(* CODESYS project SPT_Base_Types.library
   Version: 4.0.4
   Title: SPT Base Types
   DefaultNamespace: SPT_BaseTypes
   Placeholder: SPT Base Types
   Company: Beckhoff Automation LLC

Project tree, tasks and I/O mapping:
  libraries: SPT Event Logger, * (Beckhoff Automation LLC); Tc2_EtherCAT, * (Beckhoff Automation GmbH); Tc2_Standard, * (Beckhoff Automation GmbH); Tc2_System, * (Beckhoff Automation GmbH); Tc2_Utilities, * (Beckhoff Automation GmbH); Tc3_EventLogger, * (Beckhoff Automation GmbH); Tc3_JsonXml, * (Beckhoff Automation GmbH); Tc3_Module, * (Beckhoff Automation GmbH); Tc3_PackML_V3, * (Beckhoff Automation GmbH)
  Component Base/
    HMI/
      data type ST_ComponentBase_Command
      data type ST_ComponentBase_Config
      data type ST_ComponentBase_HMI
      data type ST_ComponentBase_Status
    function block FB_ComponentBase [ST]: AllowHMIControl, BlockHMIControl, Reset, CurrentAlarmSeverity, InSimulation, Name, ParentResponseDefinitions, CyclicLogic, CreateEvents, HMICommunication, Initialize, Monitoring, RaiseAlarm, RaiseAlarmWithStrings, RaiseEventWithStrings
  Framework Base/
    function block FB_BaseFB [ST]: Busy, Error, ErrorID, Marker, Trace, TraceWithJson
    function block FB_CyclicFB [ST]: CyclicLogic, InitComplete
  Interfaces/
    interface I_BaseFB: Busy, Error, ErrorID
    interface I_ComponentBase: AllowHMIControl, BlockHMIControl, Reset, CurrentAlarmSeverity, InSimulation, Name, ParentResponseDefinitions
    interface I_CyclicFB: CyclicLogic, InitComplete
    interface I_PackML_BaseModule: CurrentAlarmSeverity, DisableSubModuleModeChange, LogModeChanges, LogStateChanges, Name, ParentResponseDefinitions
    interface I_PackML_Control: ChangeMode, ChangeState, CurrentMode, CurrentState, ModeCommand, StateCommand
    interface I_PackML_ExternalController: Control, ModeChanged, StateChanged
  PackML/
    ControlSource/
      function block FB_ControlSource [ST]: CyclicLogic, Control, ModeChanged, StateChanged, Initialize, Registered
      data type ST_PackML_Control
      data type ST_PackML_Control_Simplified
    DUT/
      data type E_AlarmResponse
      data type E_PMLUnitMode
      data type ST_AvailableStateCommands
      data type ST_PackML_SubUnitInfoExt
    HMI/
      data type ST_PackMLBaseModule_Command
      data type ST_PackMLBaseModule_Config
      data type ST_PackMLBaseModule_HMI
      data type ST_PackMLBaseModule_Status
    function block FB_NextAvailablePackMLCommands [ST]: GetCommands, StateCommands
    function block FB_PackML_BaseModule [ST]: CyclicLogic, CurrentAlarmSeverity, DisableSubModuleModeChange, LogModeChanges, LogStateChanges, Name, ParentResponseDefinitions, ChangeMode, ChangeState, CurrentMode, CurrentState, ModeCommand, StateCommand, AbortImmediate, AbortImmediateError, HoldControlled, HoldImmediate, StopControlled, StopImmediate, SuspendControlled, SuspendImmediate, RaiseAlarmWithStrings, AllowHMIControl, BlockHMIControl, HMICommunication, HMIPermissions, ComponentMonitor, SubModuleMonitor, Aborted, Completed, Execute, Held, Idle, Stopped, Suspended, Undefined, ModeControl, StateControl, Aborting, Clearing, Completing, Holding, Resetting, Starting, Stopping, Suspending, Unholding, Unsuspending, CreateEvents, Initialize, ModeChanged, RegisterComponent, RegisterExternalController, RegisterSubmodule, StateChanged, StateComplete
    function block FB_PackML_ModeLogger [ST]
    function block FB_PackML_StateLogger [ST]
  Project Information/
    function F_GetCompany [ST]
    function F_GetTitle [ST]
    function F_GetVersion [ST]
  Tracing/
    function block FB_TraceLog [ST]: AddContext, AddEntry, AddEntryWithJson, FB_init, TracingAllowed
    global variables Tracing
  Version/
    global variables Global_Version
  VISUs/
    visualisation V_MachineModule
    visualisation V_Module
  text list GlobalTextList
  00000000-0000-0000-0000-000000000000|LICENSE
  LICENSE
  global variables Parameters_BaseComponent
  global variables Parameters_PackML_Base
  global variables Parameters_Tracing
*)

// Component Base/HMI/ST_ComponentBase_Command
{attribute 'OPC.UA.DA' := '1'}
{attribute 'OPC.UA.DA.StructuredType' := '1'}
{attribute 'OPC.UA.DA.Access' := '3'}
TYPE ST_ComponentBase_Command :
	STRUCT
		SimulatedOperation : BOOL;
		StandardOperation  : BOOL;
		Reset			   : BOOL;
	END_STRUCT
END_TYPE

// Component Base/HMI/ST_ComponentBase_Config
{attribute 'OPC.UA.DA' := '1'}
{attribute 'OPC.UA.DA.StructuredType' := '1'}
{attribute 'OPC.UA.DA.Access' := '1'}
TYPE ST_ComponentBase_Config :
	STRUCT
		Name : STRING;
	END_STRUCT
END_TYPE

// Component Base/HMI/ST_ComponentBase_HMI
{attribute 'OPC.UA.DA' := '1'}
{attribute 'OPC.UA.DA.StructuredType' := '1'}
TYPE ST_ComponentBase_HMI :
	STRUCT
		Config	: ST_ComponentBase_Config;
		Command : ST_ComponentBase_Command;
		Status	: ST_ComponentBase_Status;
	END_STRUCT
END_TYPE

// Component Base/HMI/ST_ComponentBase_Status
{attribute 'OPC.UA.DA' := '1'}
{attribute 'OPC.UA.DA.StructuredType' := '1'}
{attribute 'OPC.UA.DA.Access' := '1'}
TYPE ST_ComponentBase_Status :
	STRUCT
		InSimulation		: BOOL;
		Busy				: BOOL;
		Error				: BOOL;
		ErrorID				: UDINT;
		HMIControlAvailable : BOOL; // Set TRUE *FROM PLC* when HMI requests can be processed
	END_STRUCT
END_TYPE

// PackML/ControlSource/ST_PackML_Control
TYPE ST_PackML_Control :
	STRUCT
		CurrentMode		 : E_PMLUnitMode;
		ModeCommand		 : E_PMLUnitMode;
		CurrentState	 : E_PMLState;
		StateCommand	 : E_PMLCommand;
		ModeNames		 : ARRAY[0..31] OF STRING;
		ModeCommandLast	 : E_PMLUnitMode;
		StateCommandLast : E_PMLCommand;
	END_STRUCT
END_TYPE

// PackML/ControlSource/ST_PackML_Control_Simplified
TYPE ST_PackML_Control_Simplified :
	STRUCT
		ResetPermissive		: BOOL;
		StartPermissive		: BOOL;
		StopPermissive		: BOOL;
		ResetPressed AT %I* : BOOL;
		StartPressed AT %I* : BOOL;
		StopPressed	 AT %I* : BOOL;
	END_STRUCT
END_TYPE

// PackML/DUT/E_AlarmResponse
// Defines the reaction behavior to a fault
{attribute 'qualified_only'}
{attribute 'strict'}
TYPE E_AlarmResponse : (
		Abort_ImmediateError,
		Abort_Immediate,
		Stop_Immediate,
		Stop_Controlled,
		Hold_Immediate,
		Hold_Controlled,
		Suspend_Immediate,
		Suspend_Controlled,
		NoResponse
	);
END_TYPE

// PackML/DUT/E_PMLUnitMode
// Defines the allowable PackML modes  
TYPE E_PMLUnitMode : (
		Invalid		:= 0,
		Production	:= 1,
		Maintenance := 2,
		Manual		:= 3,
		UserMode1	:= 4,
		UserMode2	:= 5,
		UserMode3	:= 6,
		UserMode4	:= 7,
		UserMode5	:= 8,
		UserMode6	:= 9,
		UserMode7	:= 10,
		UserMode8	:= 11,
		UserMode9	:= 12,
		UserMode10	:= 13,
		UserMode11	:= 14,
		UserMode12	:= 15,
		UserMode13	:= 16,
		UserMode14	:= 17,
		UserMode15	:= 18,
		UserMode16	:= 19,
		UserMode17	:= 20,
		UserMode18	:= 21,
		UserMode19	:= 22,
		UserMode20	:= 23,
		UserMode21	:= 24,
		UserMode22	:= 25,
		UserMode23	:= 26,
		UserMode24	:= 27,
		UserMode25	:= 28,
		UserMode26	:= 29,
		UserMode27	:= 30,
		UserMode28	:= 31
	) DINT;
END_TYPE

// PackML/DUT/ST_AvailableStateCommands
TYPE ST_AvailableStateCommands :
	STRUCT
		Abort	  : BOOL;
		Clear	  : BOOL;
		Complete  : BOOL;
		Hold	  : BOOL;
		Reset	  : BOOL;
		Start	  : BOOL;
		Stop	  : BOOL;
		Suspend	  : BOOL;
		Unhold	  : BOOL;
		Unsuspend : BOOL;
	END_STRUCT
END_TYPE

// PackML/DUT/ST_PackML_SubUnitInfoExt
TYPE ST_PackML_SubUnitInfoExt EXTENDS ST_PMLSubUnitInfo : // Extended Struct of ST_PMLSubUnitInfo
	STRUCT
		ModuleID		: DINT;	  // Machine ID for messaging and Identification
		ModuleName		: STRING; // Human readable machine name for messaging
		UnitModeCurrent : E_PMLProtectedUnitMode;
		ActiveAlarm		: BOOL;
	END_STRUCT
END_TYPE

// PackML/HMI/ST_PackMLBaseModule_Command
{attribute 'OPC.UA.DA' := '1'}
{attribute 'OPC.UA.DA.StructuredType' := '1'}
{attribute 'OPC.UA.DA.Access' := '3'}
TYPE ST_PackMLBaseModule_Command :
	STRUCT
		Mode			   : E_PMLUnitMode				:= Parameters_PackML_Base.UNIT_MODE_DEFAULT;
		State			   : Tc3_PackML_V3.E_PMLCommand := Parameters_PackML_Base.UNIT_STATE_DEFAULT;
		ActivateStateLog   : BOOL; // HMI requests to enable the module
		DeactivateStateLog : BOOL; // HMI requests to disable the module
		ActivateModeLog	   : BOOL; // HMI requests to enable the module
		DeactivatModeLog   : BOOL; // HMI requests to disable the module
	END_STRUCT
END_TYPE

// PackML/HMI/ST_PackMLBaseModule_Config
{attribute 'OPC.UA.DA' := '1'}
{attribute 'OPC.UA.DA.StructuredType' := '1'}
{attribute 'OPC.UA.DA.Access' := '1'}
TYPE ST_PackMLBaseModule_Config :
	STRUCT
		Name			: STRING;		// Human-readable module name for user-side messaging
		LogStateChanges : BOOL := TRUE; // Toggle to permit or suppress state change logging (Should be tied to HMI setting to optionally reduce event logger clutter)
		LogModeChanges	: BOOL := TRUE; // Toggle to permit or suppress state change logging (Should be tied to HMI setting to optionally reduce event logger clutter)
		ModeNames		: ARRAY[0..31] OF STRING;
	END_STRUCT
END_TYPE

// PackML/HMI/ST_PackMLBaseModule_HMI
{attribute 'OPC.UA.DA' := '1'}
{attribute 'OPC.UA.DA.StructuredType' := '1'}
TYPE ST_PackMLBaseModule_HMI :
	STRUCT
		Config	: ST_PackMLBaseModule_Config;
		Command : ST_PackMLBaseModule_Command;
		Status	: ST_PackMLBaseModule_Status;
	END_STRUCT
END_TYPE

// PackML/HMI/ST_PackMLBaseModule_Status
{attribute 'OPC.UA.DA' := '1'}
{attribute 'OPC.UA.DA.StructuredType' := '1'}
{attribute 'OPC.UA.DA.Access' := '1'}
TYPE ST_PackMLBaseModule_Status :
	STRUCT
		Busy				: BOOL;
		Error				: BOOL;
		ErrorID				: UDINT;
		Mode				: E_PMLUnitMode;
		State				: Tc3_PackML_V3.E_PMLState;
		HMIControlAvailable : BOOL;
		StateCommands		: ST_AvailableStateCommands;
	END_STRUCT
END_TYPE

// Tracing/Tracing
{attribute 'qualified_only'}
VAR_GLOBAL
	GlobalTraceLog : FB_TraceLog;
END_VAR

// Version/Global_Version
{attribute 'TcGenerated'}
{attribute 'no-analysis'}
{attribute 'linkalways'}
// This function has been automatically generated from the project information.
VAR_GLOBAL CONSTANT
	{attribute 'const_non_replaced'}
	stLibVersion_SPT_Base_Types : ST_LibVersion := (iMajor := 4, iMinor := 0, iBuild := 4, iRevision := 0, nFlags := 1, sVersion := '4.0.4');
END_VAR

// Parameters_BaseComponent
{attribute 'qualified_only'}
VAR_GLOBAL CONSTANT
	COMPONENT_BASE_ALARM_COUNT : UINT := 2;
	INHIBIT_SIMULATION_WARNING : BOOL := FALSE;
END_VAR

// Parameters_PackML_Base
{attribute 'qualified_only'}
VAR_GLOBAL CONSTANT
	MAX_NO_OF_SUBMODULES			  : UDINT					   := 20;
	MAX_NO_OF_COMPONENTS			  : UDINT					   := 32;
	MAX_NO_OF_EXTERNAL_CONTROLLERS	  : UDINT					   := 10;
	UNIT_MODE_DEFAULT				  : E_PMLUnitMode			   := E_PMLUnitMode.Production;
	UNIT_STATE_DEFAULT				  : Tc3_PackML_V3.E_PMLCommand := E_PMLCommand.Abort;
	CONCAT_SUBMODULE_NAME_WITH_PARENT : BOOL					   := FALSE;
	CONCAT_COMPONENT_NAME_WITH_PARENT : BOOL					   := TRUE;
	SUBMODULE_NAME_DELIMETER		  : STRING(10)				   := ' ';
	COMPONENT_NAME_DELIMETER		  : STRING(10)				   := ' ';
	STATELOGGER_DISABLED			  : BOOL					   := FALSE;
	RESET_COMPONENTS_WITHOUT_ERROR	  : BOOL					   := FALSE;
	SUBSEQUENT_INIT_CALLS			  : BOOL					   := FALSE;
END_VAR

// Parameters_Tracing
{attribute 'qualified_only'}
VAR_GLOBAL CONSTANT
	TRACING_ENABLED						: BOOL	:= TRUE;
	MAX_LOG_ENTRIES_PER_SCAN			: UDINT := 100;
	ALLOW_DUPLICATE_SEQUENTIAL_MESSAGES : BOOL	:= FALSE;
END_VAR

// Component Base/FB_ComponentBase
// Basic framework of a component
FUNCTION_BLOCK ABSTRACT FB_ComponentBase EXTENDS FB_CyclicFB IMPLEMENTS I_ComponentBase
VAR
	// I_ComponentBase internal property variables
	_CurrentAlarmSeverity			: TcEventSeverity;
	_Name							: STRING; // String name of the component
	_ParentFaultResponseDefinitions : ARRAY[0..4] OF E_AlarmResponse := [E_AlarmResponse.NoResponse, E_AlarmResponse.NoResponse, E_AlarmResponse.NoResponse, E_AlarmResponse.Abort_ImmediateError, E_AlarmResponse.Abort_ImmediateError];
	_Simulate						: BOOL; // TRUE disables all hardware I/O and simulates input and output behavior

	// Alarming
	ComponentBaseAlarms : ARRAY[1..Parameters_BaseComponent.COMPONENT_BASE_ALARM_COUNT] OF FB_TcAlarm;

	// HMI Monitoring and control structure
	ComponentBase_HMI			: ST_ComponentBase_HMI;
	HMICommand_RT				: R_TRIG;
	HMICommandActive_Base		: BOOL;
	HMICommandActive_Descendant : BOOL;
END_VAR

// Sets permissive bit to allow HMI control of component functions
METHOD PUBLIC AllowHMIControl

// This method is called as required by the parent module of this component
ComponentBase_HMI.Status.HMIControlAvailable := TRUE;
END_METHOD

// Clears permissive bit to allow HMI control of component functions
METHOD PUBLIC BlockHMIControl

// This method is called as required by the parent module of this component
ComponentBase_HMI.Status.HMIControlAvailable := FALSE;
END_METHOD

// Clears error flags and error IDs for this component
METHOD PUBLIC Reset : BOOL
// This may or may not be called depending on the component type which derives FB_ComponentBase
F_ClearAllEventsInClass(ComponentBaseAlarms);
Reset := TRUE;
END_METHOD

// Returns the current alarm severity for this component
PROPERTY CurrentAlarmSeverity : TcEventSeverity
GET
CurrentAlarmSeverity := _CurrentAlarmSeverity;
END_GET
END_PROPERTY

// Enable/Disable simulation logic for this component
PROPERTY InSimulation : BOOL
GET
InSimulation := _Simulate;
END_GET
SET
_Simulate := InSimulation;
END_SET
END_PROPERTY

// Get/Set this component's name
PROPERTY Name : STRING
GET
Name := _Name;
END_GET
SET
_Name := Name;
END_SET
END_PROPERTY

PROPERTY ParentResponseDefinitions : ARRAY[0..4] OF E_AlarmResponse
GET
ParentResponseDefinitions[TcEventSeverity.Verbose]	:= _ParentFaultResponseDefinitions[TcEventSeverity.Verbose];
ParentResponseDefinitions[TcEventSeverity.Info]		:= _ParentFaultResponseDefinitions[TcEventSeverity.Info];
ParentResponseDefinitions[TcEventSeverity.Warning]	:= _ParentFaultResponseDefinitions[TcEventSeverity.Warning];
ParentResponseDefinitions[TcEventSeverity.Error]	:= _ParentFaultResponseDefinitions[TcEventSeverity.Error];
ParentResponseDefinitions[TcEventSeverity.Critical] := _ParentFaultResponseDefinitions[TcEventSeverity.Critical];
END_GET
SET
_ParentFaultResponseDefinitions[TcEventSeverity.Verbose]  := ParentResponseDefinitions[TcEventSeverity.Verbose];
_ParentFaultResponseDefinitions[TcEventSeverity.Info]	  := ParentResponseDefinitions[TcEventSeverity.Info];
_ParentFaultResponseDefinitions[TcEventSeverity.Warning]  := ParentResponseDefinitions[TcEventSeverity.Warning];
_ParentFaultResponseDefinitions[TcEventSeverity.Error]	  := ParentResponseDefinitions[TcEventSeverity.Error];
_ParentFaultResponseDefinitions[TcEventSeverity.Critical] := ParentResponseDefinitions[TcEventSeverity.Critical];
END_SET
END_PROPERTY

// This method serves as the entry point for all underlying FB logic
METHOD PUBLIC CyclicLogic

// This method should be called cyclically by descendant function blocks by invoking SUPER^.CyclicLogic().  Alternatively, the contents of this method could be reimplemented entirely in which case a call to this method would not be necessary.
IF NOT _InitComplete THEN
	_InitComplete := Initialize();
	RETURN;
END_IF

Monitoring();		// Constant error and status monitoring
HMICommunication(); // Keeps the HMI data up to date, and processes requests from the HMI for this component
END_METHOD

// Initializes event function blocks using this components's name
METHOD PROTECTED CreateEvents

// This method is called by Initialize() as required
F_CreateAllEventsInClass(Alarms		:= ComponentBaseAlarms,
						 ClassSize	:= SIZEOF(TC_EVENTS.ComponentBase),
						 pInitEvent := ADR(TC_EVENTS.ComponentBase.InitReferenceEvent),
						 Prefix		:= _Name);
END_METHOD

// Provides interlocks for HMI control and updates HMI status information for this component
METHOD PROTECTED HMICommunication

// This method is called cyclically by CyclicLogic()
//xtend this method in extended FBs to communicate specific implementation data
// Process HMI requests
HMICommand_RT(CLK := (ComponentBase_HMI.Status.HMIControlAvailable AND NOT HMICommandActive_Descendant) AND (ComponentBase_HMI.Command.Reset XOR ComponentBase_HMI.Command.SimulatedOperation XOR ComponentBase_HMI.Command.StandardOperation));

// Desendant components should observe this to interlock HMI commands
HMICommandActive_Base := ComponentBase_HMI.Status.HMIControlAvailable AND (ComponentBase_HMI.Command.Reset OR ComponentBase_HMI.Command.SimulatedOperation OR ComponentBase_HMI.Command.StandardOperation);
IF HMICommand_RT.Q THEN
	IF ComponentBase_HMI.Command.Reset THEN
		Reset();
	END_IF

	IF ComponentBase_HMI.Command.SimulatedOperation THEN
		_Simulate := TRUE;
	END_IF

	IF ComponentBase_HMI.Command.StandardOperation THEN
		_Simulate := FALSE;
	END_IF
END_IF

//pdate HMI status info
ComponentBase_HMI.Config.Name		  := _Name;
ComponentBase_HMI.Status.Busy		  := _Busy;
ComponentBase_HMI.Status.Error		  := _Error;
ComponentBase_HMI.Status.InSimulation := _Simulate;
ComponentBase_HMI.Status.ErrorID	  := _ErrorID;
END_METHOD

// Basic component initialization logic
METHOD PROTECTED Initialize : BOOL;

// This method is called by CyclicLogic() as required
// Extend initialize as needed in extended FBs
CreateEvents();
Initialize := TRUE;
END_METHOD

// Provides basic error detection and event handling for this component
METHOD PROTECTED Monitoring

// This method is called cyclically by CyclicLogic()
// Extend from extended FB with monitoring logic
IF NOT ComponentBaseAlarms[E_ComponentBase.SimulationWarning].bRaised AND _Simulate AND NOT Parameters_BaseComponent.INHIBIT_SIMULATION_WARNING THEN
	ComponentBaseAlarms[E_ComponentBase.SimulationWarning].Raise(0);
ELSIF ComponentBaseAlarms[E_ComponentBase.SimulationWarning].bRaised AND NOT _Simulate THEN
	ComponentBaseAlarms[E_ComponentBase.SimulationWarning].Clear(0, 0);
END_IF

_CurrentAlarmSeverity := TcEventSeverity.Verbose;
_CurrentAlarmSeverity := F_GetMaxSeverityRaised(Alarms := ComponentBaseAlarms, CurrentSeverity := _CurrentAlarmSeverity);
END_METHOD

// Raise an alarm, passing the faulted FB's error ID as a paramter
METHOD PROTECTED RaiseAlarm
VAR_IN_OUT
	Alarm : FB_TcAlarm;
END_VAR
F_RaiseAlarm(Alarm := Alarm);
END_METHOD

// Raises an alarm and passes string arguments as parameters for extra fault context/info
METHOD PROTECTED RaiseAlarmWithStrings
VAR_IN_OUT
	Alarm : FB_TcAlarm; // Alarm to be raised
END_VAR

VAR_INPUT
	String_1 : STRING; // First string parameter (The Name of this component will be applied first automatically)
	String_2 : STRING; // Second string parameter
END_VAR
F_RaiseAlarmWithStringsAndFlags(Alarm	  := Alarm,
								ErrorFlag := _Error,
								ErrorID	  := _ErrorID,
								String_1  := _Name,
								String_2  := String_1,
								String_3  := String_2);
END_METHOD

// Raises an alarm and passes string arguments as parameters for extra fault context/info
METHOD PROTECTED RaiseEventWithStrings
VAR_IN_OUT
	Alarm : FB_TcAlarm; // Alarm to be raised
END_VAR

VAR_INPUT
	String_1 : STRING; // First string parameter (The Name of this component will be applied first automatically)
	String_2 : STRING; // Second string parameter
END_VAR
F_RaiseAlarmWithStringParameters(Alarm	  := Alarm,
								 String_1 := _Name,
								 String_2 := String_1,
								 String_3 := String_2);
END_METHOD

END_FUNCTION_BLOCK

// Framework Base/FB_CyclicFB
FUNCTION_BLOCK ABSTRACT FB_CyclicFB EXTENDS FB_BaseFB IMPLEMENTS I_CyclicFB
VAR
	_InitComplete : BOOL;
END_VAR

// Derivatives of FB_CyclicFB should *NOT* have code in the function block body

// Use CyclicLogic() instead

METHOD PUBLIC ABSTRACT CyclicLogic
VAR_INPUT
END_VAR
END_METHOD

PROPERTY InitComplete : BOOL
GET
InitComplete := _InitComplete;
END_GET
END_PROPERTY

END_FUNCTION_BLOCK

// Framework Base/FB_BaseFB
{attribute 'reflection'}
FUNCTION_BLOCK ABSTRACT FB_BaseFB IMPLEMENTS I_BaseFB
VAR
	{attribute 'instance-path'}
	{attribute 'noinit'}
	InstancePath : STRING;
END_VAR

// I_BaseFB
VAR
	_Busy	 : BOOL := TRUE;
	_Error	 : BOOL;
	_ErrorID : UDINT;
END_VAR

// Derivatives of FB_BaseFB can have code in the function block body

PROPERTY Busy : BOOL
GET
Busy := _Busy;
END_GET
END_PROPERTY

PROPERTY Error : BOOL
GET
Error := _Error;
END_GET
END_PROPERTY

PROPERTY ErrorID : UDINT
GET
ErrorID := _ErrorID;
END_GET
END_PROPERTY

METHOD PUBLIC Marker
VAR_INPUT
	Message : T_MaxString;
END_VAR
Tracing.GlobalTraceLog.AddEntry(InstancePath, Message, 1);
END_METHOD

METHOD PUBLIC Trace
VAR_INPUT
	Message : T_MaxString;
END_VAR
Tracing.GlobalTraceLog.AddEntry(InstancePath, Message, 0);
END_METHOD

METHOD PUBLIC TraceWithJson
VAR_INPUT
	Message : T_MaxString;
	Json	: T_MaxString;
END_VAR
Tracing.GlobalTraceLog.AddEntryWithJson(InstancePath,
										Message,
										0,
										Json);
END_METHOD

END_FUNCTION_BLOCK

// Interfaces/I_BaseFB
INTERFACE I_BaseFB EXTENDS __SYSTEM.IQueryInterface

PROPERTY Busy : BOOL
GET
END_GET
END_PROPERTY

PROPERTY Error : BOOL
GET
END_GET
END_PROPERTY

PROPERTY ErrorID : UDINT;
GET
END_GET
END_PROPERTY

END_INTERFACE

// Interfaces/I_CyclicFB
INTERFACE I_CyclicFB EXTENDS I_BaseFB

METHOD CyclicLogic
VAR_INPUT
END_VAR
END_METHOD

PROPERTY InitComplete : BOOL
GET
END_GET
END_PROPERTY

END_INTERFACE

// Interfaces/I_ComponentBase
INTERFACE I_ComponentBase EXTENDS I_CyclicFB

METHOD PUBLIC AllowHMIControl
VAR_INPUT
END_VAR
END_METHOD

METHOD PUBLIC BlockHMIControl
VAR_INPUT
END_VAR
END_METHOD

METHOD PUBLIC Reset : BOOL
END_METHOD

PROPERTY CurrentAlarmSeverity : TcEventSeverity
GET
END_GET
END_PROPERTY

PROPERTY InSimulation : BOOL
GET
END_GET
SET
END_SET
END_PROPERTY

PROPERTY Name : STRING
GET
END_GET
SET
END_SET
END_PROPERTY

PROPERTY ParentResponseDefinitions : ARRAY[0..4] OF E_AlarmResponse
GET
END_GET
SET
END_SET
END_PROPERTY

END_INTERFACE

// Interfaces/I_PackML_BaseModule
INTERFACE I_PackML_BaseModule EXTENDS I_CyclicFB, I_PackML_Control

PROPERTY CurrentAlarmSeverity : TcEventSeverity
GET
END_GET
END_PROPERTY

PROPERTY DisableSubModuleModeChange : BOOL
GET
END_GET
SET
END_SET
END_PROPERTY

PROPERTY LogModeChanges : BOOL
GET
END_GET
SET
END_SET
END_PROPERTY

PROPERTY LogStateChanges : BOOL
GET
END_GET
SET
END_SET
END_PROPERTY

PROPERTY Name : STRING
GET
END_GET
SET
END_SET
END_PROPERTY

PROPERTY ParentResponseDefinitions : ARRAY[0..4] OF E_AlarmResponse
GET
END_GET
SET
END_SET
END_PROPERTY

END_INTERFACE

// Interfaces/I_PackML_Control
INTERFACE I_PackML_Control

METHOD ChangeMode
VAR_INPUT
	Mode : E_PMLUnitMode;
END_VAR
END_METHOD

METHOD ChangeState
VAR_INPUT
	State : E_PMLCommand;
END_VAR
END_METHOD

PROPERTY CurrentMode : E_PMLUnitMode
GET
END_GET
END_PROPERTY

PROPERTY CurrentState : E_PMLState
GET
END_GET
END_PROPERTY

PROPERTY ModeCommand : DINT
GET
END_GET
SET
END_SET
END_PROPERTY

PROPERTY StateCommand : E_PMLCommand
GET
END_GET
SET
END_SET
END_PROPERTY

END_INTERFACE

// Interfaces/I_PackML_ExternalController
INTERFACE I_PackML_ExternalController

PROPERTY Control : I_PackML_Control
SET
END_SET
END_PROPERTY

METHOD ModeChanged
VAR_INPUT
	NewMode : E_PMLUnitMode;
END_VAR
END_METHOD

METHOD StateChanged
VAR_INPUT
	NewState : E_PMLCommand;
END_VAR
END_METHOD

END_INTERFACE

// PackML/ControlSource/FB_ControlSource
FUNCTION_BLOCK FB_ControlSource EXTENDS FB_CyclicFB IMPLEMENTS I_PackML_ExternalController
VAR
	ipModule				  : I_PackML_Control;
	MainPMLControl_Simplified : ST_PackML_Control_Simplified;
	MainPMLControl_Standard	  : ST_PackML_Control;
	R_HMICommand			  : R_TRIG;
END_VAR

METHOD CyclicLogic
VAR
	i : UDINT;
END_VAR
IF NOT _InitComplete THEN
	_InitComplete := Initialize();
	RETURN;
END_IF

// Copy the module to the local mode and state
MainPMLControl_Standard.CurrentMode	 := ipModule.CurrentMode;
MainPMLControl_Standard.CurrentState := ipModule.CurrentState;
FOR i := 1 TO 5 DO
	MainPMLControl_Standard.ModeNames[i] := F_PMLUnitModeToString(TO_DINT(i));
END_FOR

// Process requests
R_HMICommand(CLK := (MainPMLControl_Simplified.ResetPressed XOR MainPMLControl_Simplified.StartPressed XOR MainPMLControl_Simplified.StopPressed) XOR (MainPMLControl_Standard.StateCommand <> E_PMLCommand.Undefined AND MainPMLControl_Standard.StateCommandLast <> MainPMLControl_Standard.StateCommand) XOR (MainPMLControl_Standard.ModeCommandLast <> MainPMLControl_Standard.ModeCommand));
IF R_HMICommand.Q THEN
	MainPMLControl_Standard.ModeCommandLast	 := MainPMLControl_Standard.ModeCommand;
	MainPMLControl_Standard.StateCommandLast := MainPMLControl_Standard.StateCommand;
	IF MainPMLControl_Simplified.ResetPressed AND MainPMLControl_Simplified.ResetPermissive AND MainPMLControl_Standard.CurrentState = E_PMLState.Aborted THEN
		ipModule.ChangeState(Tc3_PackML_V3.E_PMLCommand.Clear);
	ELSIF MainPMLControl_Simplified.ResetPressed AND MainPMLControl_Simplified.ResetPermissive THEN
		ipModule.ChangeState(Tc3_PackML_V3.E_PMLCommand.Reset);
	ELSIF MainPMLControl_Simplified.StartPressed AND MainPMLControl_Simplified.StartPermissive THEN
		IF MainPMLControl_Standard.CurrentState = Tc3_PackML_V3.E_PMLState.Idle THEN
			ipModule.ChangeState(Tc3_PackML_V3.E_PMLCommand.Start);
		ELSIF MainPMLControl_Standard.CurrentState = Tc3_PackML_V3.E_PMLState.Held THEN
			ipModule.ChangeState(Tc3_PackML_V3.E_PMLCommand.Unhold);
		END_IF
	ELSIF MainPMLControl_Simplified.StopPressed AND MainPMLControl_Simplified.StopPermissive THEN
		ipModule.ChangeState(Tc3_PackML_V3.E_PMLCommand.Stop);
	ELSIF ipModule.StateCommand <> MainPMLControl_Standard.StateCommand THEN
		ipModule.StateCommand := MainPMLControl_Standard.StateCommand;
	ELSIF ipModule.ModeCommand <> MainPMLControl_Standard.ModeCommand THEN
		ipModule.ModeCommand := MainPMLControl_Standard.ModeCommand;
	END_IF
END_IF

// Set the permissives for each button
MainPMLControl_Simplified.StartPermissive := MainPMLControl_Standard.CurrentState = Tc3_PackML_V3.E_PMLState.Idle OR MainPMLControl_Standard.CurrentState = Tc3_PackML_V3.E_PMLState.Held;
MainPMLControl_Simplified.StopPermissive  :=
	(MainPMLControl_Standard.CurrentState <> Tc3_PackML_V3.E_PMLState.Stopped AND MainPMLControl_Standard.CurrentState <> Tc3_PackML_V3.E_PMLState.Clearing AND MainPMLControl_Standard.CurrentState <> Tc3_PackML_V3.E_PMLState.Aborted AND MainPMLControl_Standard.CurrentState <> Tc3_PackML_V3.E_PMLState.Aborting AND MainPMLControl_Standard.CurrentState <> Tc3_PackML_V3.E_PMLState.Undefined);

MainPMLControl_Simplified.ResetPermissive := MainPMLControl_Standard.CurrentState = Tc3_PackML_V3.E_PMLState.Completed OR MainPMLControl_Standard.CurrentState = Tc3_PackML_V3.E_PMLState.Stopped OR MainPMLControl_Standard.CurrentState = Tc3_PackML_V3.E_PMLState.Aborted;
END_METHOD

PROPERTY Control : I_PackML_Control
SET
ipModule := Control;
END_SET
END_PROPERTY

METHOD FINAL ModeChanged
VAR_INPUT
	NewMode : E_PMLUnitMode;
END_VAR
MainPMLControl_Standard.ModeCommand := NewMode;
END_METHOD

METHOD FINAL StateChanged
VAR_INPUT
	NewState : E_PMLCommand;
END_VAR
MainPMLControl_Standard.StateCommand := NewState;
END_METHOD

METHOD FINAL Initialize : BOOL
IF Registered THEN
	Initialize := TRUE;
END_IF
END_METHOD

PROPERTY Registered : BOOL
GET
Registered := ipModule <> 0;
END_GET
END_PROPERTY

END_FUNCTION_BLOCK

// PackML/FB_NextAvailablePackMLCommands
FUNCTION_BLOCK FB_NextAvailablePackMLCommands
VAR
	NextAvailableCommands : ARRAY[1..MAX_AVAILABLE_COMMANDS] OF E_PMLCommand;
	i					  : DINT;
END_VAR

VAR //Property Backers
	_StateCommands : ST_AvailableStateCommands;
END_VAR

VAR CONSTANT
	MAX_AVAILABLE_COMMANDS : DINT := 10;
END_VAR

METHOD PUBLIC GetCommands : ARRAY[1..10] OF E_PMLCommand
VAR_INPUT
	CurrentMode	 : E_PMLUnitMode;
	CurrentState : E_PMLState;
END_VAR

VAR
	ModeConfiguration : Tc3_PackML_V3.ST_PMLUnitModeConfiguration;
END_VAR
FOR i := 1 TO MAX_AVAILABLE_COMMANDS DO
	NextAvailableCommands[i] := E_PMLCommand.Undefined;
END_FOR

_StateCommands.Abort	 := FALSE;
_StateCommands.Clear	 := FALSE;
_StateCommands.Complete	 := FALSE;
_StateCommands.Hold		 := FALSE;
_StateCommands.Reset	 := FALSE;
_StateCommands.Start	 := FALSE;
_StateCommands.Stop		 := FALSE;
_StateCommands.Suspend	 := FALSE;
_StateCommands.Unhold	 := FALSE;
_StateCommands.Unsuspend := FALSE;
i						 := 1;
ModeConfiguration		 := Tc3_PackML_V3.GlobalVariables.stPMLUnitModeConfiguration[CurrentMode];
// Generate next possible Commands
CASE CurrentState OF
	E_PMLState.Undefined:
		;

	E_PMLState.Aborting:
		;

	E_PMLState.Aborted:
		NextAvailableCommands[i] := E_PMLCommand.Clear;
		_StateCommands.Clear	 := TRUE;

	E_PMLState.Clearing:
		;

	E_PMLState.Stopping:
		NextAvailableCommands[i] := E_PMLCommand.Abort;
		_StateCommands.Abort	 := TRUE;

	E_PMLState.Stopped:
		NextAvailableCommands[i] := E_PMLCommand.Abort;
		_StateCommands.Abort	 := TRUE;
		i						 := i + 1;
		IF NOT ModeConfiguration.aStateDisabled[E_PMLState.Resetting] AND NOT ModeConfiguration.aStateDisabled[E_PMLState.Idle] THEN
			NextAvailableCommands[i] := E_PMLCommand.Reset;
			_StateCommands.Reset	 := TRUE;
		ELSE
			NextAvailableCommands[i] := E_PMLCommand.Start;
			_StateCommands.Start	 := TRUE;
		END_IF

	E_PMLState.Resetting:
		NextAvailableCommands[i] := E_PMLCommand.Abort;
		_StateCommands.Abort	 := TRUE;
		i						 := i + 1;
		NextAvailableCommands[i] := E_PMLCommand.Stop;
		_StateCommands.Stop		 := TRUE;

	E_PMLState.Idle:
		NextAvailableCommands[i] := E_PMLCommand.Abort;
		_StateCommands.Abort	 := TRUE;
		i						 := i + 1;
		NextAvailableCommands[i] := E_PMLCommand.Stop;
		_StateCommands.Stop		 := TRUE;
		i						 := i + 1;
		NextAvailableCommands[i] := E_PMLCommand.Start;
		_StateCommands.Start	 := TRUE;

	E_PMLState.Starting:
		NextAvailableCommands[i] := E_PMLCommand.Abort;
		_StateCommands.Abort	 := TRUE;
		i						 := i + 1;
		NextAvailableCommands[i] := E_PMLCommand.Stop;
		_StateCommands.Stop		 := TRUE;

	E_PMLState.Execute:
		NextAvailableCommands[i] := E_PMLCommand.Abort;
		_StateCommands.Abort	 := TRUE;
		i						 := i + 1;
		NextAvailableCommands[i] := E_PMLCommand.Stop;
		_StateCommands.Stop		 := TRUE;
		i						 := i + 1;
		IF (NOT ModeConfiguration.aStateDisabled[E_PMLState.Held] AND NOT ModeConfiguration.aStateDisabled[E_PMLState.Holding]) OR (NOT ModeConfiguration.aStateDisabled[E_PMLState.Held] AND NOT ModeConfiguration.aStateDisabled[E_PMLState.Unholding]) THEN
			NextAvailableCommands[i] := E_PMLCommand.Hold;
			_StateCommands.Hold		 := TRUE;
			i						 := i + 1;
		END_IF

		IF (NOT ModeConfiguration.aStateDisabled[E_PMLState.Suspended] AND NOT ModeConfiguration.aStateDisabled[E_PMLState.Suspending]) OR (NOT ModeConfiguration.aStateDisabled[E_PMLState.Suspended] AND NOT ModeConfiguration.aStateDisabled[E_PMLState.Unsuspending]) THEN
			NextAvailableCommands[i] := E_PMLCommand.Suspend;
			_StateCommands.Suspend	 := TRUE;
			i						 := i + 1;
		END_IF

		IF NOT ModeConfiguration.aStateDisabled[E_PMLState.Completed] AND NOT ModeConfiguration.aStateDisabled[E_PMLState.Completing] THEN
			NextAvailableCommands[i] := E_PMLCommand.Complete;
			_StateCommands.Complete	 := TRUE;
		END_IF

	E_PMLState.Completing:
		NextAvailableCommands[i] := E_PMLCommand.Abort;
		_StateCommands.Abort	 := TRUE;
		i						 := i + 1;
		NextAvailableCommands[i] := E_PMLCommand.Stop;
		_StateCommands.Stop		 := TRUE;

	E_PMLState.Completed:
		NextAvailableCommands[i] := E_PMLCommand.Abort;
		_StateCommands.Abort	 := TRUE;
		i						 := i + 1;
		NextAvailableCommands[i] := E_PMLCommand.Stop;
		_StateCommands.Stop		 := TRUE;
		i						 := i + 1;
		IF NOT ModeConfiguration.aStateDisabled[E_PMLState.Resetting] AND NOT ModeConfiguration.aStateDisabled[E_PMLState.Idle] THEN
			NextAvailableCommands[i] := E_PMLCommand.Reset;
			_StateCommands.Reset	 := TRUE;
		ELSE
			NextAvailableCommands[i] := E_PMLCommand.Start;
			_StateCommands.Start	 := TRUE;
		END_IF

	E_PMLState.Holding:
		NextAvailableCommands[i] := E_PMLCommand.Abort;
		_StateCommands.Abort	 := TRUE;
		i						 := i + 1;
		NextAvailableCommands[i] := E_PMLCommand.Stop;
		_StateCommands.Stop		 := TRUE;

	E_PMLState.Held:
		NextAvailableCommands[i] := E_PMLCommand.Abort;
		_StateCommands.Abort	 := TRUE;
		i						 := i + 1;
		NextAvailableCommands[i] := E_PMLCommand.Stop;
		_StateCommands.Stop		 := TRUE;
		i						 := i + 1;
		NextAvailableCommands[i] := E_PMLCommand.Unhold;
		_StateCommands.Unhold	 := TRUE;
		i						 := i + 1;
		IF NOT ModeConfiguration.aStateDisabled[E_PMLState.Completed] AND NOT ModeConfiguration.aStateDisabled[E_PMLState.Completing] THEN
			NextAvailableCommands[i] := E_PMLCommand.Complete;
			_StateCommands.Complete	 := TRUE;
		END_IF

	E_PMLState.Unholding:
		NextAvailableCommands[i] := E_PMLCommand.Abort;
		_StateCommands.Abort	 := TRUE;
		i						 := i + 1;
		NextAvailableCommands[i] := E_PMLCommand.Stop;
		_StateCommands.Stop		 := TRUE;

	E_PMLState.Suspending:
		NextAvailableCommands[i] := E_PMLCommand.Abort;
		_StateCommands.Abort	 := TRUE;
		i						 := i + 1;
		NextAvailableCommands[i] := E_PMLCommand.Stop;
		_StateCommands.Stop		 := TRUE;

	E_PMLState.Suspended:
		NextAvailableCommands[i] := E_PMLCommand.Abort;
		_StateCommands.Abort	 := TRUE;
		i						 := i + 1;
		NextAvailableCommands[i] := E_PMLCommand.Stop;
		_StateCommands.Stop		 := TRUE;
		i						 := i + 1;
		NextAvailableCommands[i] := E_PMLCommand.Unsuspend;
		_StateCommands.Unsuspend := TRUE;
		i						 := i + 1;
		IF NOT ModeConfiguration.aStateDisabled[E_PMLState.Completed] AND NOT ModeConfiguration.aStateDisabled[E_PMLState.Completing] THEN
			NextAvailableCommands[i] := E_PMLCommand.Complete;
			_StateCommands.Complete	 := TRUE;
			i						 := i + 1;
		END_IF

		IF (NOT ModeConfiguration.aStateDisabled[E_PMLState.Held] AND NOT ModeConfiguration.aStateDisabled[E_PMLState.Holding]) OR (NOT ModeConfiguration.aStateDisabled[E_PMLState.Held] AND NOT ModeConfiguration.aStateDisabled[E_PMLState.Unholding]) THEN
			NextAvailableCommands[i] := E_PMLCommand.Hold;
			_StateCommands.Hold		 := TRUE;
		END_IF

	E_PMLState.Unsuspending:
		NextAvailableCommands[i] := E_PMLCommand.Abort;
		_StateCommands.Abort	 := TRUE;
		i						 := i + 1;
		NextAvailableCommands[i] := E_PMLCommand.Stop;
		_StateCommands.Stop		 := TRUE;
END_CASE

GetCommands := NextAvailableCommands;
END_METHOD

PROPERTY StateCommands : REFERENCE TO ST_AvailableStateCommands
GET
StateCommands REF= _StateCommands;
END_GET
END_PROPERTY

END_FUNCTION_BLOCK

// PackML/FB_PackML_BaseModule
FUNCTION_BLOCK ABSTRACT FB_PackML_BaseModule EXTENDS FB_CyclicFB IMPLEMENTS I_PackML_BaseModule, I_PackML_Control
VAR
	_CurrentMode	: E_PMLUnitMode; // Current UnitMode of the module	
	_CommandedMode	: E_PMLUnitMode; // Current Commanded UnitMode of the module
	_CurrentState	: Tc3_PackML_V3.E_PMLState;
	_CommandedState : Tc3_PackML_V3.E_PMLCommand;
END_VAR

VAR
	_CurrentAlarmSeverity			: TcEventSeverity;
	_LogModeChanges					: BOOL := TRUE;	 // Toggle to permit or suppress state change logging (Should be tied to HMI setting to optionally reduce event logger clutter)
	_LogStateChanges				: BOOL := FALSE; // Toggle to permit or suppress state change logging (Should be tied to HMI setting to optionally reduce event logger clutter)
	_DisableSubModuleModeChange		: BOOL := FALSE; // Disable the Automatic Mode Change of all SubModules on Mode Change for this PML instanz
	_Name							: STRING;		 // Human-readable module name for user-side messaging
	_ParentFaultResponseDefinitions : ARRAY[0..4] OF E_AlarmResponse := [E_AlarmResponse.NoResponse, E_AlarmResponse.NoResponse, E_AlarmResponse.NoResponse, E_AlarmResponse.Abort_ImmediateError, E_AlarmResponse.Abort_ImmediateError];
END_VAR

VAR
	ModeManager						  : FB_PMLUnitModeManager; // Manages operating mode transitions and rules
	StateMachine					  : FB_PMLStateMachine;	   // Manages PackML state transitions
	CustomModes						  : FB_PMLUnitModeConfig;  // Used to define custom machine modes if desired
	PMLStateLogger					  : FB_PackML_StateLogger; // Logs PackML state changes
	PMLModeLogger					  : FB_PackML_ModeLogger;  // Logs PackML Mode changes	
	AvailablePackMLCommands			  : FB_NextAvailablePackMLCommands;
	PackMLBaseModule_HMI			  : ST_PackMLBaseModule_HMI;	// Handles status and control communications with the HMI
	PMLSubModuleInfoRef				  : ST_PMLSubUnitInfoRef;		// Reference to the subunit information, used by the state machine
	LastModeCommand					  : E_PMLUnitMode;				// Previous received PackML mode command
	LastMode						  : DINT;						// Last PackML mode 	
	LastState						  : Tc3_PackML_V3.E_PMLState;	// Last cycle PackML state
	StateTasksComplete				  : BOOL := FALSE;				// All tasks to be performed at this program level are complete
	NoStateTasksToComplete			  : BOOL := TRUE;				// Indicates whether this stateneeds to perform tasks other than commanding its children
	PackMLAlarms					  : ARRAY[1..48] OF FB_TcAlarm; // Array of alarms for PackML state and mode changes that exist in any PackML enabled module
	BaseAlarms						  : ARRAY[1..32] OF FB_TcAlarm; // Array of alarms for general module Alarms				
	ipSubModules					  : ARRAY[1..Parameters_PackML_Base.MAX_NO_OF_SUBMODULES] OF I_PackML_BaseModule;
	PMLSubModuleInfo				  : ARRAY[1..Parameters_PackML_Base.MAX_NO_OF_SUBMODULES] OF ST_PMLSubUnitInfo;
	NumberOfSubModules				  : UDINT := 0; // calculated number of instantiated sub modules
	ipComponents					  : ARRAY[1..Parameters_PackML_Base.MAX_NO_OF_COMPONENTS] OF I_ComponentBase;
	NumberOfComponents				  : UDINT := 0; // calculated number of instantiated components
	ModeNames						  : ARRAY[0..31] OF STRING;
	ipExternalControllers			  : ARRAY[1..Parameters_PackML_Base.MAX_NO_OF_EXTERNAL_CONTROLLERS] OF I_PackML_ExternalController;
	ReachedInitialDefaultStateAndMode : BOOL;
	ModeChangeRequested				  : BOOL;
	SequenceState					  : UDINT;
	DescendantSequenceState			  : UDINT;
	HMICommand_RT					  : R_TRIG;
	HMICommandActive_Base			  : BOOL;
	HMICommandActive_Descendant		  : BOOL;
	CurrentNextAvailableCommands	  : ARRAY[1..10] OF E_PMLCommand;
END_VAR

//*********************************************************

// !!!!! Code implementation only in CyclicLogic() method !!!!! 

//*********************************************************

// This method serves as the entry point for all underlying FB logic

// This method should be called cyclically by descendant function blocks by invoking SUPER^.CyclicLogic().  Alternatively, the contents of this method could be reimplemented entirely in which case a call to this method would not be necessary.
METHOD PUBLIC CyclicLogic
VAR
	i : UDINT;
END_VAR
//*********************************************************

// If you are about to write actual machine implementation code, note that implementation code should exist within an implementation machine module block that extends this machine module base!

//*********************************************************
// Descendents of this FB which override this methods should use SUPER^.Initialize()
IF NOT _InitComplete THEN
	_InitComplete := Initialize();
	RETURN;
END_IF

// Inhibit mode & state errors until startup is complete
IF NOT ReachedInitialDefaultStateAndMode AND _CurrentState = E_PMLState.Aborted AND _CurrentMode = Parameters_PackML_Base.UNIT_MODE_DEFAULT THEN
	ReachedInitialDefaultStateAndMode := TRUE;
END_IF

// Call this module's subunits, if any are defined
FOR i := 1 TO NumberOfSubModules DO
	IF ipSubModules[i] <> 0 THEN
		ipSubModules[i].CyclicLogic();
		PMLSubModuleInfo[i].eState := ipSubModules[i].CurrentState; // Reflect the state of the subunits to the state machine of the module		
	END_IF
END_FOR

FOR i := 1 TO NumberOfComponents DO
	IF ipComponents[i] <> 0 THEN
		ipComponents[i].CyclicLogic();
	END_IF
END_FOR

// Handle HMI communications--this must happen before state control!!
HMICommunication();

// Mode control loop of the module
ModeControl();

// State control loop of the module
StateControl();

//
SubModuleMonitor();
ComponentMonitor();
HMIPermissions();

//
CurrentNextAvailableCommands						:= AvailablePackMLCommands.GetCommands(_CurrentMode, _CurrentState);
PackMLBaseModule_HMI.Status.StateCommands.Abort		:= AvailablePackMLCommands.StateCommands.Abort;
PackMLBaseModule_HMI.Status.StateCommands.Reset		:= AvailablePackMLCommands.StateCommands.Reset;
PackMLBaseModule_HMI.Status.StateCommands.Start		:= AvailablePackMLCommands.StateCommands.Start;
PackMLBaseModule_HMI.Status.StateCommands.Stop		:= AvailablePackMLCommands.StateCommands.Stop;
PackMLBaseModule_HMI.Status.StateCommands.Hold		:= AvailablePackMLCommands.StateCommands.Hold;
PackMLBaseModule_HMI.Status.StateCommands.Unhold	:= AvailablePackMLCommands.StateCommands.Unhold;
PackMLBaseModule_HMI.Status.StateCommands.Suspend	:= AvailablePackMLCommands.StateCommands.Suspend;
PackMLBaseModule_HMI.Status.StateCommands.Unsuspend := AvailablePackMLCommands.StateCommands.Unsuspend;
PackMLBaseModule_HMI.Status.StateCommands.Clear		:= AvailablePackMLCommands.StateCommands.Clear;
PackMLBaseModule_HMI.Status.StateCommands.Complete	:= AvailablePackMLCommands.StateCommands.Complete;

//
_CurrentAlarmSeverity := TcEventSeverity.Verbose;
_CurrentAlarmSeverity := F_GetMaxSeverityRaised(Alarms := PackMLAlarms, CurrentSeverity := _CurrentAlarmSeverity);
_CurrentAlarmSeverity := F_GetMaxSeverityRaised(Alarms := BaseAlarms, CurrentSeverity := _CurrentAlarmSeverity);
END_METHOD

// Returns the highest severity of any event(s) currently raised 
PROPERTY CurrentAlarmSeverity : TcEventSeverity
GET
CurrentAlarmSeverity := _CurrentAlarmSeverity;
END_GET
END_PROPERTY

// Disable the Automatic Mode Change of all SubModules on Mode Change for this PML instanz
PROPERTY DisableSubModuleModeChange : BOOL
GET
DisableSubModuleModeChange := _DisableSubModuleModeChange;
END_GET
SET
_DisableSubModuleModeChange := DisableSubModuleModeChange;
END_SET
END_PROPERTY

// Enable/Disable logging of mode changes
PROPERTY LogModeChanges : BOOL
GET
LogModeChanges := _LogModeChanges;
END_GET
SET
_LogModeChanges := LogModeChanges;
END_SET
END_PROPERTY

// Enable/Disable logging of state changes
PROPERTY LogStateChanges : BOOL
GET
LogStateChanges := _LogStateChanges;
END_GET
SET
_LogStateChanges := LogStateChanges;
END_SET
END_PROPERTY

// Get/Set the name of this module
PROPERTY Name : STRING
GET
Name := _Name;
END_GET
SET
_Name := Name;
END_SET
END_PROPERTY

PROPERTY ParentResponseDefinitions : ARRAY[0..4] OF E_AlarmResponse
GET
ParentResponseDefinitions[TcEventSeverity.Verbose]	:= _ParentFaultResponseDefinitions[TcEventSeverity.Verbose];
ParentResponseDefinitions[TcEventSeverity.Info]		:= _ParentFaultResponseDefinitions[TcEventSeverity.Info];
ParentResponseDefinitions[TcEventSeverity.Warning]	:= _ParentFaultResponseDefinitions[TcEventSeverity.Warning];
ParentResponseDefinitions[TcEventSeverity.Error]	:= _ParentFaultResponseDefinitions[TcEventSeverity.Error];
ParentResponseDefinitions[TcEventSeverity.Critical] := _ParentFaultResponseDefinitions[TcEventSeverity.Critical];
END_GET
SET
_ParentFaultResponseDefinitions[TcEventSeverity.Verbose]  := ParentResponseDefinitions[TcEventSeverity.Verbose];
_ParentFaultResponseDefinitions[TcEventSeverity.Info]	  := ParentResponseDefinitions[TcEventSeverity.Info];
_ParentFaultResponseDefinitions[TcEventSeverity.Warning]  := ParentResponseDefinitions[TcEventSeverity.Warning];
_ParentFaultResponseDefinitions[TcEventSeverity.Error]	  := ParentResponseDefinitions[TcEventSeverity.Error];
_ParentFaultResponseDefinitions[TcEventSeverity.Critical] := ParentResponseDefinitions[TcEventSeverity.Critical];
END_SET
END_PROPERTY

METHOD ChangeMode
VAR_INPUT
	Mode : E_PMLUnitMode;
END_VAR
IF Mode <> _CommandedMode THEN
	ModeCommand := Mode;
END_IF
END_METHOD

METHOD ChangeState
VAR_INPUT
	State : E_PMLCommand;
END_VAR
IF State <> _CommandedState THEN
	StateCommand := State;
END_IF
END_METHOD

// Returns the current PackML mode of this module
PROPERTY CurrentMode : E_PMLUnitMode
GET
CurrentMode := _CurrentMode;
END_GET
END_PROPERTY

// Returns current PackML state of this module
PROPERTY CurrentState : Tc3_PackML_V3.E_PMLState
GET
CurrentState := _CurrentState;
END_GET
END_PROPERTY

// Sets the requested PackML Mode
PROPERTY ModeCommand : DINT
GET
ModeCommand := _CommandedMode;
END_GET
SET
VAR
	i : UDINT;
END_VAR
IF ModeCommand <> _CommandedMode THEN
	_CommandedMode					  := ModeCommand;
	PackMLBaseModule_HMI.Command.Mode := ModeCommand;
	// Notify external controllers that state has changed	
	FOR i := 1 TO Parameters_PackML_Base.MAX_NO_OF_EXTERNAL_CONTROLLERS DO
		IF ipExternalControllers[i] <> 0 THEN
			ipExternalControllers[i].ModeChanged(_CommandedMode);
		END_IF
	END_FOR
END_IF
END_SET
END_PROPERTY

// Sets the requested PackML state
PROPERTY StateCommand : Tc3_PackML_V3.E_PMLCommand
GET
StateCommand := _CommandedState;
END_GET
SET
VAR
	i : UDINT;
END_VAR
IF _CurrentMode <> E_PMLUnitMode.Invalid AND _CurrentState <> E_PMLState.Undefined THEN
	_CommandedState					   := StateCommand;
	PackMLBaseModule_HMI.Command.State := StateCommand;
	// Notify external controllers that state has changed
	FOR i := 1 TO Parameters_PackML_Base.MAX_NO_OF_EXTERNAL_CONTROLLERS DO
		IF ipExternalControllers[i] <> 0 THEN
			ipExternalControllers[i].StateChanged(_CommandedState);
		END_IF
	END_FOR
END_IF
END_SET
END_PROPERTY

// Provides fault reaction logic where the module state is driven to the Aborting state
METHOD PROTECTED AbortImmediate

(*
No error is thrown by this fault reaction.
This method is called by ComponentMonitor() or SubModuleMonitor() as required
*)
ChangeState(E_PMLCommand.Abort);
END_METHOD

// Provides fault reaction logic where the module state is driven to the Aborting state
METHOD PROTECTED AbortImmediateError
VAR_INPUT
	Name	 : STRING; // The name of the faulting submodule or component
	IsModule : BOOL;   // If TRUE a SubModuleError is thrown.  If FALSE a ComponentError is thrown. 
END_VAR

(*
This fault reaction throws an accompanying error
This method is called by ComponentMonitor() or SubModuleMonitor() as required
*)
IF IsModule THEN
	IF NOT BaseAlarms[E_BaseAlarms.SubModuleError].bRaised THEN
		F_RaiseAlarmWithStringParameters(BaseAlarms[E_BaseAlarms.SubModuleError],
										 _Name,
										 Name,
										 '');
	END_IF
ELSE
	IF NOT BaseAlarms[E_BaseAlarms.ComponentError].bRaised THEN
		F_RaiseAlarmWithStringParameters(BaseAlarms[E_BaseAlarms.ComponentError],
										 _Name,
										 Name,
										 '');
	END_IF
END_IF

THIS^.ChangeState(E_PMLCommand.Abort);
END_METHOD

// Provides fault reaction logic where the module state is driven to the Holding state at the next available opportunity
METHOD PROTECTED HoldControlled

(*
No error is thrown by this fault reaction.
This method is called by ComponentMonitor() or SubModuleMonitor() as required
*)
ChangeState(E_PMLCommand.Hold);
END_METHOD

// Provides fault reaction logic where the module state is driven to the Holding state immediately
METHOD PROTECTED HoldImmediate

(*
No error is thrown by this fault reaction.
This method is called by <c>ComponentMonitor()</c> or <c>SubModuleMonitor()</c> as required
*)
ChangeState(E_PMLCommand.Hold);
END_METHOD

// Provides fault reaction logic where the module state is driven to the Stopping state at the next available opportunity
METHOD PROTECTED StopControlled

(*
No error is thrown by this fault reaction.
This method is called by ComponentMonitor() or SubModuleMonitor() as required
*)
ChangeState(E_PMLCommand.Stop);
END_METHOD

// Provides fault reaction logic where the module state is driven to the Stopping state immediately
METHOD PROTECTED StopImmediate

(*
No error is thrown by this fault reaction.
This method is called by ComponentMonitor() or SubModuleMonitor() as required
*)
ChangeState(E_PMLCommand.Stop);
END_METHOD

// Provides fault reaction logic where the module state is driven to the Suspending state at the next available opportunity
METHOD PROTECTED SuspendControlled

(*
No error is thrown by this fault reaction.
This method is called by ComponentMonitor() or SubModuleMonitor() as required
*)
ChangeState(E_PMLCommand.Suspend);
END_METHOD

// Provides fault reaction logic where the module state is driven to the Suspending state immediately
METHOD PROTECTED SuspendImmediate

(*
No error is thrown by this fault reaction.
This method is called by ComponentMonitor() or SubModuleMonitor() as required
*)
ChangeState(E_PMLCommand.Suspend);
END_METHOD

// Raises an alarm and passes string arguments as parameters for extra fault context/info
METHOD PROTECTED RaiseAlarmWithStrings
VAR_IN_OUT
	Alarm : FB_TcAlarm; // Alarm to be raised
END_VAR

VAR_INPUT
	String_1 : STRING; // First string parameter (The Name of this component will be applied first automatically)
	String_2 : STRING; // Second string parameter
END_VAR
F_RaiseAlarmWithStringParameters(Alarm	  := Alarm,
								 String_1 := Name,
								 String_2 := String_1,
								 String_3 := String_2);
END_METHOD

// Sets permissive bit to allow HMI control of module and component functions
METHOD PROTECTED FINAL AllowHMIControl
VAR_INPUT
	ThisModuleOnly : BOOL; // If TRUE, only the PackML module itself is controllable. If FALSE, all components become controllable as well
END_VAR

VAR
	i : UDINT;
END_VAR

// This method is called as required by the HMIPermissions() method
PackMLBaseModule_HMI.Status.HMIControlAvailable := TRUE;
IF ThisModuleOnly THEN
	FOR i := 1 TO NumberOfComponents DO
		ipComponents[i].BlockHMIControl();
	END_FOR
ELSE
	FOR i := 1 TO NumberOfComponents DO
		ipComponents[i].AllowHMIControl();
	END_FOR
END_IF
END_METHOD

// Clears permissive bit to disallow HMI control of module and component functions
METHOD PROTECTED FINAL BlockHMIControl
VAR
	i : UDINT;
END_VAR

// This method is called as required by the HMIPermissions() method
PackMLBaseModule_HMI.Status.HMIControlAvailable := FALSE;
FOR i := 1 TO NumberOfComponents DO
	ipComponents[i].BlockHMIControl();
END_FOR
END_METHOD

// Provides interlocks for HMI control and updates HMI status information for this module
METHOD PROTECTED HMICommunication

// This method is called cyclically by CyclicLogic()
// Extend this method in extended FBs to communicate specific implementation data
// Process HMI requests
HMICommand_RT(CLK := (PackMLBaseModule_HMI.Status.HMIControlAvailable AND NOT HMICommandActive_Descendant) AND
					 (PackMLBaseModule_HMI.Command.ActivateModeLog XOR PackMLBaseModule_HMI.Command.DeactivatModeLog XOR PackMLBaseModule_HMI.Command.ActivateStateLog XOR PackMLBaseModule_HMI.Command.DeactivateStateLog XOR PackMLBaseModule_HMI.Command.Mode <> _CommandedMode XOR PackMLBaseModule_HMI.Command.State <> _CommandedState));

// Desendant components should observe this to interlock HMI commands
HMICommandActive_Base := PackMLBaseModule_HMI.Status.HMIControlAvailable AND (PackMLBaseModule_HMI.Command.ActivateModeLog OR PackMLBaseModule_HMI.Command.DeactivatModeLog OR PackMLBaseModule_HMI.Command.ActivateStateLog OR PackMLBaseModule_HMI.Command.DeactivateStateLog XOR PackMLBaseModule_HMI.Command.Mode <> _CommandedMode XOR PackMLBaseModule_HMI.Command.State <> _CommandedState);
IF HMICommand_RT.Q THEN
	IF PackMLBaseModule_HMI.Command.ActivateModeLog THEN
		_LogModeChanges := TRUE;
	END_IF

	IF PackMLBaseModule_HMI.Command.DeactivatModeLog THEN
		_LogModeChanges := FALSE;
	END_IF

	IF PackMLBaseModule_HMI.Command.ActivateStateLog THEN
		_LogStateChanges := TRUE;
	END_IF

	IF PackMLBaseModule_HMI.Command.DeactivateStateLog THEN
		_LogStateChanges := FALSE;
	END_IF

	IF PackMLBaseModule_HMI.Command.Mode <> _CommandedMode THEN
		ModeCommand := PackMLBaseModule_HMI.Command.Mode;
	END_IF

	IF PackMLBaseModule_HMI.Command.State <> _CommandedState THEN
		StateCommand := PackMLBaseModule_HMI.Command.State;
	END_IF
END_IF

PackMLBaseModule_HMI.Config.Name			:= _Name;
PackMLBaseModule_HMI.Config.LogModeChanges	:= _LogModeChanges;
PackMLBaseModule_HMI.Config.LogStateChanges := _LogStateChanges;
PackMLBaseModule_HMI.Config.ModeNames		:= ModeNames;
PackMLBaseModule_HMI.Status.Mode			:= _CurrentMode;
PackMLBaseModule_HMI.Status.State			:= _CurrentState;
PackMLBaseModule_HMI.Status.Busy			:= _Busy;
PackMLBaseModule_HMI.Status.Error			:= _Error;
PackMLBaseModule_HMI.Status.ErrorID			:= _ErrorID;
END_METHOD

// Automatically enables and disables HMI control based on the PackML mode
METHOD PROTECTED HMIPermissions

// This method is called cyclically by CyclicLogic()
// General Mode Based Monitoring and handling of HMI control
CASE _CurrentMode OF
	E_PMLUnitMode.Production:
		CASE _CurrentState OF
			E_PMLState.Stopped:
				AllowHMIControl(ThisModuleOnly := TRUE); // Allow control for recovery
			E_PMLState.Idle:
				BlockHMIControl();

			E_PMLState.Suspended:
				BlockHMIControl();

			E_PMLState.Execute:
				BlockHMIControl();

			E_PMLState.Aborted:
				AllowHMIControl(ThisModuleOnly := TRUE); // Allow control for recovery
			E_PMLState.Held:
				AllowHMIControl(ThisModuleOnly := TRUE); // Allow control for recovery
			E_PMLState.Completed:
				BlockHMIControl();
		END_CASE

	E_PMLUnitMode.Manual:
		AllowHMIControl(ThisModuleOnly := FALSE);

	E_PMLUnitMode.Maintenance:
		AllowHMIControl(ThisModuleOnly := FALSE);
END_CASE
END_METHOD

// This method monitors components within this PackML module and initiates fault responses as required
METHOD PROTECTED ComponentMonitor : BOOL
VAR
	AlarmResponses : ARRAY[0..4] OF E_AlarmResponse; // Temporary response array
	i			   : UDINT;
END_VAR

// This method is called cyclically by CyclicLogic()
FOR i := 1 TO NumberOfComponents DO
	IF _CurrentState <> E_PMLState.Aborted AND _CurrentState <> E_PMLState.Aborting AND _CurrentState <> E_PMLState.Clearing AND _CurrentState <> E_PMLState.Stopped AND _CurrentState <> E_PMLState.Stopping THEN
		AlarmResponses := ipComponents[i].ParentResponseDefinitions;
		CASE AlarmResponses[ipComponents[i].CurrentAlarmSeverity] OF
			E_AlarmResponse.Abort_ImmediateError:
				AbortImmediateError(ipComponents[i].Name, FALSE);

			E_AlarmResponse.Abort_Immediate:
				AbortImmediate();

			E_AlarmResponse.Stop_Immediate:
				StopImmediate();

			E_AlarmResponse.Stop_Controlled:
				StopControlled();

			E_AlarmResponse.Hold_Immediate:
				HoldImmediate();

			E_AlarmResponse.Hold_Controlled:
				HoldControlled();

			E_AlarmResponse.Suspend_Immediate:
				SuspendImmediate();

			E_AlarmResponse.Suspend_Controlled:
				SuspendControlled();

			E_AlarmResponse.NoResponse:
				;
		END_CASE
	ELSIF _CurrentState = E_PMLState.Stopped OR _CurrentState = E_PMLState.Stopping THEN
		AlarmResponses := ipComponents[i].ParentResponseDefinitions;
		CASE AlarmResponses[ipComponents[i].CurrentAlarmSeverity] OF
			E_AlarmResponse.Abort_ImmediateError:
				AbortImmediateError(ipComponents[i].Name, FALSE);

			E_AlarmResponse.Abort_Immediate:
				AbortImmediate();

			E_AlarmResponse.NoResponse:
				;
		END_CASE
	END_IF
END_FOR
END_METHOD

// This method monitors submodules within this PackML module and initiates fault responses as required
METHOD PROTECTED SubModuleMonitor : BOOL
VAR
	AlarmResponses : ARRAY[0..4] OF E_AlarmResponse; // Temporary response array	
	i			   : UDINT;
END_VAR

// This method is called cyclically by CyclicLogic()
FOR i := 1 TO NumberOfSubModules DO
	IF _CurrentState <> E_PMLState.Aborted AND _CurrentState <> E_PMLState.Aborting AND _CurrentState <> E_PMLState.Clearing AND _CurrentState <> E_PMLState.Stopped AND _CurrentState <> E_PMLState.Stopping THEN
		AlarmResponses := ipSubModules[i].ParentResponseDefinitions;
		CASE AlarmResponses[ipSubModules[i].CurrentAlarmSeverity] OF
			E_AlarmResponse.Abort_ImmediateError:
				AbortImmediateError(ipSubModules[i].Name, TRUE);

			E_AlarmResponse.Abort_Immediate:
				AbortImmediate();

			E_AlarmResponse.Stop_Immediate:
				StopImmediate();

			E_AlarmResponse.Stop_Controlled:
				StopControlled();

			E_AlarmResponse.Hold_Immediate:
				HoldImmediate();

			E_AlarmResponse.Hold_Controlled:
				HoldControlled();

			E_AlarmResponse.Suspend_Immediate:
				SuspendImmediate();

			E_AlarmResponse.Suspend_Controlled:
				SuspendControlled();

			E_AlarmResponse.NoResponse:
				;
		END_CASE
	ELSIF _CurrentState = E_PMLState.Stopped OR _CurrentState = E_PMLState.Stopping THEN
		AlarmResponses := ipSubModules[i].ParentResponseDefinitions;
		CASE AlarmResponses[ipSubModules[i].CurrentAlarmSeverity] OF
			E_AlarmResponse.Abort_ImmediateError:
				AbortImmediateError(ipSubModules[i].Name, TRUE);

			E_AlarmResponse.Abort_Immediate:
				AbortImmediate();

			E_AlarmResponse.NoResponse:
				;
		END_CASE
	END_IF
END_FOR
END_METHOD

// This method contains code which will execute when this PackML module is in the Aborted state
METHOD PROTECTED Aborted

(*
The base implementation of this method is empty. User must override this method to provide functionality.
This method is called as required by StateControl()
*)
//*************************************************************************************************************************************************************************

// If you are about to write application specific code, note that any such code should exist within the "Application" directory using a Function Block that 'EXTENDS' this base Function Block!

// This particular method's functionality can be overriden in the extended block by creating a method of the same name, with desired functionality therein

// If the functionality of this base module is to be retained, but more functionality is desired, the extended method can contain a SUPER^.ThisMethodName(); call, which will call this code

//*************************************************************************************************************************************************************************
END_METHOD

// This method contains code which will execute when this PackML module is in the Complete state
METHOD PROTECTED Completed

(*
The base implementation of this method is empty. User must override this method to provide functionality.
This method is called as required by StateControl()
*)
//*************************************************************************************************************************************************************************

// If you are about to write application specific code, note that any such code should exist within the "Application" directory using a Function Block that 'EXTENDS' this base Function Block!

// This particular method's functionality can be overriden in the extended block by creating a method of the same name, with desired functionality therein

// If the functionality of this base module is to be retained, but more functionality is desired, the extended method can contain a SUPER^.ThisMethodName(); call, which will call this code

//*************************************************************************************************************************************************************************
END_METHOD

// This method contains code which will execute when this PackML module is in the Execute state
METHOD PROTECTED Execute

(*
The base implementation of this method is empty. User must override this method to provide functionality.
This method is called as required by StateControl()
*)
//*************************************************************************************************************************************************************************

// If you are about to write application specific code, note that any such code should exist within the "Application" directory using a Function Block that 'EXTENDS' this base Function Block!

// This particular method's functionality can be overriden in the extended block by creating a method of the same name, with desired functionality therein

// If the functionality of this base module is to be retained, but more functionality is desired, the extended method can contain a SUPER^.ThisMethodName(); call, which will call this code

//*************************************************************************************************************************************************************************
END_METHOD

// This method contains code which will execute when this PackML module is in the Held state
METHOD PROTECTED Held

(*
The base implementation of this method is empty. User must override this method to provide functionality.
This method is called as required by StateControl()
*)
//*************************************************************************************************************************************************************************

// If you are about to write application specific code, note that any such code should exist within the "Application" directory using a Function Block that 'EXTENDS' this base Function Block!

// This particular method's functionality can be overriden in the extended block by creating a method of the same name, with desired functionality therein

// If the functionality of this base module is to be retained, but more functionality is desired, the extended method can contain a SUPER^.ThisMethodName(); call, which will call this code

//*************************************************************************************************************************************************************************
END_METHOD

// This method contains code which will execute when this PackML module is in the Idle state
METHOD PROTECTED Idle

(*
The base implementation of this method is empty. User must override this method to provide functionality.
This method is called as required by StateControl()
*)
//*************************************************************************************************************************************************************************

// If you are about to write application specific code, note that any such code should exist within the "Application" directory using a Function Block that 'EXTENDS' this base Function Block!

// This particular method's functionality can be overriden in the extended block by creating a method of the same name, with desired functionality therein

// If the functionality of this base module is to be retained, but more functionality is desired, the extended method can contain a SUPER^.ThisMethodName(); call, which will call this code

//*************************************************************************************************************************************************************************
END_METHOD

// This method contains code which will execute when this PackML module is in the Stopped state
METHOD PROTECTED Stopped

(*
The base implementation of this method is empty. User must override this method to provide functionality.
This method is called as required by StateControl()
*)
//*************************************************************************************************************************************************************************

// If you are about to write application specific code, note that any such code should exist within the "Application" directory using a Function Block that 'EXTENDS' this base Function Block!

// This particular method's functionality can be overriden in the extended block by creating a method of the same name, with desired functionality therein

// If the functionality of this base module is to be retained, but more functionality is desired, the extended method can contain a SUPER^.ThisMethodName(); call, which will call this code

//*************************************************************************************************************************************************************************
END_METHOD

// This method contains code which will execute when this PackML module is in the Suspended state
METHOD PROTECTED Suspended

(*
The base implementation of this method is empty. User must override this method to provide functionality.
This method is called as required by StateControl()
*)
//*************************************************************************************************************************************************************************

// If you are about to write application specific code, note that any such code should exist within the "Application" directory using a Function Block that 'EXTENDS' this base Function Block!

// This particular method's functionality can be overriden in the extended block by creating a method of the same name, with desired functionality therein

// If the functionality of this base module is to be retained, but more functionality is desired, the extended method can contain a SUPER^.ThisMethodName(); call, which will call this code

//*************************************************************************************************************************************************************************
END_METHOD

// This method contains code which will execute when this PackML module is in a state which is not defined by the PackML standard
METHOD PROTECTED Undefined

(*
The base implementation of this method is empty. User must override this method to provide functionality.
This state should not be reached under normal circumstances.
This method is called as required by StateControl()
*)
//*************************************************************************************************************************************************************************

// If you are about to write application specific code, note that any such code should exist within the "Application" directory using a Function Block that 'EXTENDS' this base Function Block!

// This particular method's functionality can be overriden in the extended block by creating a method of the same name, with desired functionality therein

// If the functionality of this base module is to be retained, but more functionality is desired, the extended method can contain a SUPER^.ThisMethodName(); call, which will call this code

//*************************************************************************************************************************************************************************
END_METHOD

// Handles mode change requests for this module and all submodules
METHOD PRIVATE FINAL ModeControl
VAR
	i : UDINT;
END_VAR

// This method is called cyclically by CyclicLogic()
// On startup, Mode is invalid, set it to production
IF _CurrentMode = E_PMLUnitMode.Invalid THEN
	ModeChangeRequested := TRUE;
	_CommandedMode		:= Parameters_PackML_Base.UNIT_MODE_DEFAULT;
	// Notify external controllers that state has changed	
	FOR i := 1 TO Parameters_PackML_Base.MAX_NO_OF_EXTERNAL_CONTROLLERS DO
		IF ipExternalControllers[i] <> 0 THEN
			ipExternalControllers[i].ModeChanged(_CommandedMode);
		END_IF
	END_FOR

	LastModeCommand := _CommandedMode;

// If mode is valid and the command has changed, attempt to change modes
ELSIF _CommandedMode <> LastModeCommand THEN
	ModeChangeRequested				  := TRUE;
	PackMLBaseModule_HMI.Command.Mode := _CommandedMode;
	// Notify external controllers that state has changed	
	FOR i := 1 TO Parameters_PackML_Base.MAX_NO_OF_EXTERNAL_CONTROLLERS DO
		IF ipExternalControllers[i] <> 0 THEN
			ipExternalControllers[i].ModeChanged(_CommandedMode);
		END_IF
	END_FOR

	LastModeCommand := _CommandedMode;
END_IF

IF ModeChangeRequested THEN
	// Handles mode changes based on ModeCommand and the state transition rules defined in the pre-defined protected modes or custom modes
	ModeManager(bExecute	 := TRUE,
				eModeCommand := _CommandedMode,
				eState		 := _CurrentState,
				eModeStatus	 => _CurrentMode);

	IF ModeManager.bDone THEN
		IF PackMLAlarms[E_PackMLBase_Alarms.ModeCommandInvalid].bRaised THEN
			PackMLAlarms[E_PackMLBase_Alarms.ModeCommandInvalid].Clear(0, 0);
		END_IF

		// If PackML mode has changed
		IF ModeManager.eModeStatus <> LastMode THEN
			LastMode				:= ModeManager.eModeStatus;
			SequenceState			:= 0;
			DescendantSequenceState := 0;
			ModeChanged();
			// If state change logging is not suppressed
			IF _LogModeChanges THEN
				PMLModeLogger(Alarms := PackMLAlarms, ModulePrefix := _Name, Mode := ModeManager.eModeStatus);
			END_IF

			IF NOT _DisableSubModuleModeChange THEN
				// Change SubModules
				FOR i := 1 TO NumberOfSubModules DO
					ipSubModules[i].ModeCommand := ModeManager.eModeStatus; // Call the SetMode loop of the subunits 
				END_FOR
			END_IF
		END_IF

		// Reset mode control command
		ModeManager(bExecute := FALSE);
		ModeChangeRequested := FALSE;
	ELSIF ModeManager.bError THEN
		IF ReachedInitialDefaultStateAndMode THEN
			IF NOT PackMLAlarms[E_PackMLBase_Alarms.ModeCommandInvalid].bRaised THEN
				PackMLAlarms[E_PackMLBase_Alarms.ModeCommandInvalid].Raise(0);
				_CommandedMode					  := _CurrentMode;
				PackMLBaseModule_HMI.Command.Mode := _CurrentMode;
			END_IF
		END_IF

		// Reset mode control command
		ModeManager(bExecute := FALSE);
		ModeChangeRequested := FALSE;
	END_IF
END_IF
END_METHOD

// Calls PackML state manager and corresponding methods according to current module state
METHOD PRIVATE FINAL StateControl
// This method is called cyclically by CyclicLogic()
VAR
	i : UDINT;
END_VAR
// On startup, state is invalid, set it to default
IF _CurrentState = E_PMLState.Undefined AND _CurrentMode <> E_PMLUnitMode.Invalid THEN
	_CommandedState := Parameters_PackML_Base.UNIT_STATE_DEFAULT;
END_IF

// Call PackML state machine	
StateMachine(eMode			  := _CurrentMode,
			 eCommand		  := _CommandedState,
			 stSubUnitInfoRef :=,
			 stOptions		  :=,
			 eState			  => _CurrentState,
			 sState			  =>,
			 bError			  =>,
			 nErrorID		  =>);

// If PackML state has changed
IF _CurrentState <> LastState THEN
	LastState						   := _CurrentState;
	PackMLBaseModule_HMI.Command.State := _CommandedState;
	// Notify external controllers that state has changed
	FOR i := 1 TO Parameters_PackML_Base.MAX_NO_OF_EXTERNAL_CONTROLLERS DO
		IF ipExternalControllers[i] <> 0 THEN
			ipExternalControllers[i].StateChanged(_CommandedState);
		END_IF
	END_FOR

	SequenceState			:= 0;
	DescendantSequenceState := 0;
	NoStateTasksToComplete	:= TRUE;
	StateChanged();
END_IF

IF ReachedInitialDefaultStateAndMode THEN
	// Log appropriate state changes
	IF NOT Parameters_PackML_Base.STATELOGGER_DISABLED THEN
		PMLStateLogger(Alarms		 := PackMLAlarms,
					   ModulePrefix	 := _Name,
					   State		 := _CurrentState,
					   LogAllChanges := _LogStateChanges);
	END_IF
END_IF

// Call appropriate method depending on current PackML state
CASE _CurrentState OF
	E_PMLState.Undefined:
		Undefined();

	E_PMLState.Clearing:
		Clearing();

	E_PMLState.Stopped:
		Stopped();

	E_PMLState.Starting:
		Starting();

	E_PMLState.Idle:
		Idle();

	E_PMLState.Suspended:
		Suspended();

	E_PMLState.Execute:
		Execute();

	E_PMLState.Stopping:
		Stopping();

	E_PMLState.Aborting:
		Aborting();

	E_PMLState.Aborted:
		Aborted();

	E_PMLState.Holding:
		Holding();

	E_PMLState.Held:
		Held();

	E_PMLState.Unholding:
		Unholding();

	E_PMLState.Suspending:
		Suspending();

	E_PMLState.Unsuspending:
		Unsuspending();

	E_PMLState.Resetting:
		Resetting();

	E_PMLState.Completing:
		Completing();

	E_PMLState.Completed:
		Completed();
END_CASE
END_METHOD

// This method contains code which will execute when this PackML module is in the Aborting state
METHOD PROTECTED Aborting
VAR
	i				: UDINT;
	SubModulesReady : BOOL := TRUE;
END_VAR

// Note: The Abort command should be associated with the fault handing routine of a module. It should not be directly commanded from any user inteface. 

// This method is called as required by <c>StateControl()</c>
//*************************************************************************************************************************************************************************

// If you are about to write application specific code, note that any such code should exist within the "Application" directory using a Function Block that 'EXTENDS' this base Function Block!

// This particular method's functionality can be overriden in the extended block by creating a method of the same name, with desired functionality therein

// If the functionality of this base module is to be retained, but more functionality is desired, the extended method can contain a SUPER^.ThisMethodName(); call, which will call this code

//*************************************************************************************************************************************************************************

// Perform State tasks here
// Send abort command to all sub modules
FOR i := 1 TO NumberOfSubModules DO
	ipSubModules[i].StateCommand := E_PMLCommand.Abort;
END_FOR

FOR i := 1 TO NumberOfSubModules DO
	SubModulesReady := SubModulesReady AND (ipSubModules[i].CurrentState = E_PMLState.Aborted);
END_FOR

IF SubModulesReady AND (StateTasksComplete OR NoStateTasksToComplete) THEN
	NoStateTasksToComplete := TRUE;
	StateTasksComplete	   := FALSE;
	StateComplete();
END_IF
END_METHOD

// This method contains code which will execute when this PackML module is in the Clearing state
METHOD PROTECTED Clearing
VAR
	i				: UDINT;
	SubModulesReady : BOOL := TRUE;
END_VAR

// Note: The Clear command can also be thought of as a fault reset depite the ambiguity in the naming of the Reset state. 

// This method is called as required by <c>StateControl()</c>
//*************************************************************************************************************************************************************************

// If you are about to write application specific code, note that any such code should exist within the "Application" directory using a Function Block that 'EXTENDS' this base Function Block!

// This particular method's functionality can be overriden in the extended block by creating a method of the same name, with desired functionality therein

// If the functionality of this base module is to be retained, but more functionality is desired, the extended method can contain a SUPER^.ThisMethodName(); call, which will call this code

//*************************************************************************************************************************************************************************

// Perform State tasks here
// Send clear command to all sub modules
FOR i := 1 TO NumberOfSubModules DO
	ipSubModules[i].StateCommand := E_PMLCommand.Clear;
END_FOR

IF BaseAlarms[E_BaseAlarms.ComponentError].bRaised THEN
	BaseAlarms[E_BaseAlarms.ComponentError].Clear(0, 0);
END_IF;

IF BaseAlarms[E_BaseAlarms.SubModuleError].bRaised THEN
	BaseAlarms[E_BaseAlarms.SubModuleError].Clear(0, 0);
END_IF;

FOR i := 1 TO NumberOfComponents DO
	IF Parameters_PackML_Base.RESET_COMPONENTS_WITHOUT_ERROR THEN
		ipComponents[i].Reset();
	ELSE
		IF ipComponents[i].Error THEN
			ipComponents[i].Reset();
		END_IF
	END_IF
END_FOR

FOR i := 1 TO NumberOfComponents DO
	SubModulesReady := SubModulesReady AND NOT ipComponents[i].Error;
END_FOR

FOR i := 1 TO NumberOfSubModules DO
	SubModulesReady := SubModulesReady AND (ipSubModules[i].CurrentState = E_PMLState.Stopped);
END_FOR

IF SubModulesReady AND (StateTasksComplete OR NoStateTasksToComplete) THEN
	NoStateTasksToComplete := TRUE;
	StateTasksComplete	   := FALSE;
	StateComplete();
END_IF
END_METHOD

// This method contains code which will execute when this PackML module is in the Completing state
METHOD PROTECTED Completing
VAR
	i				: UDINT;
	SubModulesReady : BOOL := TRUE;
END_VAR

// This method is called as required by <c>StateControl()</c>
//*************************************************************************************************************************************************************************

// If you are about to write application specific code, note that any such code should exist within the "Application" directory using a Function Block that 'EXTENDS' this base Function Block!

// This particular method's functionality can be overriden in the extended block by creating a method of the same name, with desired functionality therein

// If the functionality of this base module is to be retained, but more functionality is desired, the extended method can contain a SUPER^.ThisMethodName(); call, which will call this code

//*************************************************************************************************************************************************************************

// Perform State tasks here
// Send complete command to all sub modules
FOR i := 1 TO NumberOfSubModules DO
	ipSubModules[i].StateCommand := E_PMLCommand.Complete;
END_FOR

FOR i := 1 TO NumberOfSubModules DO
	SubModulesReady := SubModulesReady AND (ipSubModules[i].CurrentState = E_PMLState.Completed);
END_FOR

IF SubModulesReady AND (StateTasksComplete OR NoStateTasksToComplete) THEN
	NoStateTasksToComplete := TRUE;
	StateTasksComplete	   := FALSE;
	StateComplete();
END_IF
END_METHOD

// This method contains code which will execute when this PackML module is in the Holding state
METHOD PROTECTED Holding
VAR
	i				: UDINT;
	SubModulesReady : BOOL := TRUE;
END_VAR

// Note: The Hold command is intended to be given by an operator. It is meant to be distinct from a Suspend in that upstream/downstream jams, etc. should be handled automatically using Suspend.  Both Hold and Suspend result in a paused state which should allow resumption of the Execute state. 

// This method is called as required by StateControl()
//*************************************************************************************************************************************************************************

// If you are about to write application specific code, note that any such code should exist within the "Application" directory using a Function Block that 'EXTENDS' this base Function Block!

// This particular method's functionality can be overriden in the extended block by creating a method of the same name, with desired functionality therein

// If the functionality of this base module is to be retained, but more functionality is desired, the extended method can contain a SUPER^.ThisMethodName(); call, which will call this code

//*************************************************************************************************************************************************************************

// Perform State tasks here
// Send hold command to all sub modules
FOR i := 1 TO NumberOfSubModules DO
	ipSubModules[i].StateCommand := E_PMLCommand.Hold;
END_FOR

FOR i := 1 TO NumberOfSubModules DO
	SubModulesReady := SubModulesReady AND (ipSubModules[i].CurrentState = E_PMLState.Held);
END_FOR

IF SubModulesReady AND (StateTasksComplete OR NoStateTasksToComplete) THEN
	NoStateTasksToComplete := TRUE;
	StateTasksComplete	   := FALSE;
	StateComplete();
END_IF
END_METHOD

// This method contains code which will execute when this PackML module is in the Resetting state
METHOD PROTECTED Resetting
VAR
	i				: UDINT;
	SubModulesReady : BOOL := TRUE;
END_VAR

// Note: The Reset command can also be thought of as an enable depite the ambiguity in the naming of the Clearing state.

// This method is called as required by StateControl()
//*************************************************************************************************************************************************************************

// If you are about to write application specific code, note that any such code should exist within the "Application" directory using a Function Block that 'EXTENDS' this base Function Block!

// This particular method's functionality can be overriden in the extended block by creating a method of the same name, with desired functionality therein

// If the functionality of this base module is to be retained, but more functionality is desired, the extended method can contain a SUPER^.ThisMethodName(); call, which will call this code

//*************************************************************************************************************************************************************************

// Perform State tasks here

// Send clear/reset command to all sub modules
// As long as this module is in the "Resetting" state, it will attempt to get all modules to Idle by sending abort, clear, and reset commands as appropriate to its children until they do
FOR i := 1 TO NumberOfSubModules DO
	IF ipSubModules[i].CurrentState = E_PMLState.Stopped OR ipSubModules[i].CurrentState = E_PMLState.Completed THEN
		ipSubModules[i].StateCommand := E_PMLCommand.Reset;
	ELSIF ipSubModules[i].CurrentState = E_PMLState.Aborted THEN
		ipSubModules[i].StateCommand := E_PMLCommand.Clear;
	ELSIF ipSubModules[i].CurrentState = E_PMLState.Clearing OR ipSubModules[i].CurrentState = E_PMLState.Stopping OR ipSubModules[i].CurrentState = E_PMLState.Resetting OR ipSubModules[i].CurrentState = E_PMLState.Idle THEN
		;
	ELSE
		ipSubModules[i].StateCommand := E_PMLCommand.Abort;
	END_IF
END_FOR

FOR i := 1 TO NumberOfSubModules DO
	SubModulesReady := SubModulesReady AND (ipSubModules[i].CurrentState = E_PMLState.Idle);
END_FOR

IF SubModulesReady AND (StateTasksComplete OR NoStateTasksToComplete) THEN
	NoStateTasksToComplete := TRUE;
	StateTasksComplete	   := FALSE;
	StateComplete();
END_IF
END_METHOD

// This method contains code which will execute when this PackML module is in the Starting state
METHOD PROTECTED Starting
VAR
	i				: UDINT;
	SubModulesReady : BOOL := TRUE;
END_VAR

// This method is called as required by StateControl()
//*************************************************************************************************************************************************************************

// If you are about to write application specific code, note that any such code should exist within the "Application" directory using a Function Block that 'EXTENDS' this base Function Block!

// This particular method's functionality can be overriden in the extended block by creating a method of the same name, with desired functionality therein

// If the functionality of this base module is to be retained, but more functionality is desired, the extended method can contain a SUPER^.ThisMethodName(); call, which will call this code

//*************************************************************************************************************************************************************************

// Perform State tasks here
// Send start command to all sub modules
FOR i := 1 TO NumberOfSubModules DO
	ipSubModules[i].StateCommand := E_PMLCommand.Start;
END_FOR

FOR i := 1 TO NumberOfSubModules DO
	SubModulesReady := SubModulesReady AND (ipSubModules[i].CurrentState = E_PMLState.Execute);
END_FOR

IF SubModulesReady AND (StateTasksComplete OR NoStateTasksToComplete) THEN
	NoStateTasksToComplete := TRUE;
	StateTasksComplete	   := FALSE;
	StateComplete();
END_IF
END_METHOD

// This method contains code which will execute when this PackML module is in the Stopping state
METHOD PROTECTED Stopping
VAR
	i				: UDINT;
	SubModulesReady : BOOL := TRUE;
END_VAR

// This method is called as required by StateControl()
//*************************************************************************************************************************************************************************

// If you are about to write application specific code, note that any such code should exist within the "Application" directory using a Function Block that 'EXTENDS' this base Function Block!

// This particular method's functionality can be overriden in the extended block by creating a method of the same name, with desired functionality therein

// If the functionality of this base module is to be retained, but more functionality is desired, the extended method can contain a SUPER^.ThisMethodName(); call, which will call this code

//*************************************************************************************************************************************************************************

// Perform State tasks here
// Send stop command to all sub modules
FOR i := 1 TO NumberOfSubModules DO
	ipSubModules[i].StateCommand := E_PMLCommand.Stop;
END_FOR

FOR i := 1 TO NumberOfSubModules DO
	SubModulesReady := SubModulesReady AND (ipSubModules[i].CurrentState = E_PMLState.Stopped OR ipSubModules[i].CurrentState = E_PMLState.Aborted);
END_FOR

IF SubModulesReady AND (StateTasksComplete OR NoStateTasksToComplete) THEN
	NoStateTasksToComplete := TRUE;
	StateTasksComplete	   := FALSE;
	StateComplete();
END_IF
END_METHOD

// This method contains code which will execute when this PackML module is in the Suspending state
METHOD PROTECTED Suspending
VAR
	i				: UDINT;
	SubModulesReady : BOOL := TRUE;
END_VAR

// Note: The Suspend command is intended to be initiated by automatic detection of upstream/downstream jams, etc. It is meant to be distinct from a Hold in that Hold should be commanded by an operator.  Both Hold and Suspend result in a paused state which should allow resumption of the Execute state. 

// This method is called as required by StateControl()
//*************************************************************************************************************************************************************************

// If you are about to write application specific code, note that any such code should exist within the "Application" directory using a Function Block that 'EXTENDS' this base Function Block!

// This particular method's functionality can be overriden in the extended block by creating a method of the same name, with desired functionality therein

// If the functionality of this base module is to be retained, but more functionality is desired, the extended method can contain a SUPER^.ThisMethodName(); call, which will call this code

//*************************************************************************************************************************************************************************

//Perform State tasks here
// Send suspend command to all sub modules
FOR i := 1 TO NumberOfSubModules DO
	ipSubModules[i].StateCommand := E_PMLCommand.Suspend;
END_FOR

FOR i := 1 TO NumberOfSubModules DO
	SubModulesReady := SubModulesReady AND (ipSubModules[i].CurrentState = E_PMLState.Suspended);
END_FOR

IF SubModulesReady AND (StateTasksComplete OR NoStateTasksToComplete) THEN
	NoStateTasksToComplete := TRUE;
	StateTasksComplete	   := FALSE;
	StateComplete();
END_IF
END_METHOD

// This method contains code which will execute when this PackML module is in the Unholding state
METHOD PROTECTED Unholding
VAR
	i				: UDINT;
	SubModulesReady : BOOL := TRUE;
END_VAR

// This method is called as required by <c>StateControl()</c>
//*************************************************************************************************************************************************************************

// If you are about to write application specific code, note that any such code should exist within the "Application" directory using a Function Block that 'EXTENDS' this base Function Block!

// This particular method's functionality can be overriden in the extended block by creating a method of the same name, with desired functionality therein

// If the functionality of this base module is to be retained, but more functionality is desired, the extended method can contain a SUPER^.ThisMethodName(); call, which will call this code

//*************************************************************************************************************************************************************************

// Perform State tasks here
// Send unhold command to all sub modules
FOR i := 1 TO NumberOfSubModules DO
	ipSubModules[i].StateCommand := E_PMLCommand.Unhold;
END_FOR

FOR i := 1 TO NumberOfSubModules DO
	SubModulesReady := SubModulesReady AND (ipSubModules[i].CurrentState = E_PMLState.Execute);
END_FOR

IF SubModulesReady AND (StateTasksComplete OR NoStateTasksToComplete) THEN
	NoStateTasksToComplete := TRUE;
	StateTasksComplete	   := FALSE;
	StateComplete();
END_IF
END_METHOD

// This method contains code which will execute when this PackML module is in the Unsuspending state
METHOD PROTECTED Unsuspending
VAR
	i				: UDINT;
	SubModulesReady : BOOL := TRUE;
END_VAR

// This method is called as required by StateControl()
//*************************************************************************************************************************************************************************

// If you are about to write application specific code, note that any such code should exist within the "Application" directory using a Function Block that 'EXTENDS' this base Function Block!

// This particular method's functionality can be overriden in the extended block by creating a method of the same name, with desired functionality therein

// If the functionality of this base module is to be retained, but more functionality is desired, the extended method can contain a SUPER^.ThisMethodName(); call, which will call this code

//*************************************************************************************************************************************************************************

// Perform State tasks here
// Send unsuspend command to all sub modules
FOR i := 1 TO NumberOfSubModules DO
	ipSubModules[i].StateCommand := E_PMLCommand.Unsuspend;
END_FOR

FOR i := 1 TO NumberOfSubModules DO
	SubModulesReady := SubModulesReady AND (ipSubModules[i].CurrentState = E_PMLState.Execute);
END_FOR

IF SubModulesReady AND (StateTasksComplete OR NoStateTasksToComplete) THEN
	NoStateTasksToComplete := TRUE;
	StateTasksComplete	   := FALSE;
	StateComplete();
END_IF
END_METHOD

// Initializes event function blocks using this module's name
METHOD PROTECTED CreateEvents

// This method is called by Initialize() as required
F_CreateAllEventsInClass(Alarms		:= PackMLAlarms,
						 ClassSize	:= SIZEOF(TC_EVENTS.PackMLBase_Alarms),
						 pInitEvent := ADR(TC_EVENTS.PackMLBase_Alarms.InitReferenceEvent),
						 Prefix		:= _Name);

F_CreateAllEventsInClass(Alarms		:= BaseAlarms,
						 ClassSize	:= SIZEOF(TC_EVENTS.BaseAlarms),
						 pInitEvent := ADR(TC_EVENTS.BaseAlarms.InitReferenceEvent),
						 Prefix		:= _Name);
END_METHOD

// Basic module initialization logic
METHOD PROTECTED Initialize : BOOL;
VAR
	i						 : UDINT;
	varInfo					 : __SYSTEM.VAR_INFO;
	AllSubUnitsInitialized	 : BOOL := TRUE;
	AllComponentsInitialized : BOOL := TRUE;
END_VAR

VAR_INST
	c, m : UDINT;
END_VAR

// This method is called by CyclicLogic() as required
// This method may get called several times while waiting for subunits/components to init so it makes sense to break it up into a state machine
CASE SequenceState OF
	0:
		CreateEvents();
		c			  := 1;
		m			  := 1;
		SequenceState := SequenceState + 10;

	10:
		// Figure out how many Submodules were instantiated - they should be from 1 to X and not skip any indices.
		NumberOfSubModules := 0;
		FOR i := 1 TO Parameters_PackML_Base.MAX_NO_OF_SUBMODULES DO
			IF ipSubModules[i] <> 0 THEN
				NumberOfSubModules		   := NumberOfSubModules + 1;
				PMLSubModuleInfo[i].Active := TRUE; // Follows Main State Machine
				IF Parameters_PackML_Base.CONCAT_SUBMODULE_NAME_WITH_PARENT THEN
					ipSubModules[i].Name := CONCAT(CONCAT(_Name, Parameters_PackML_Base.SUBMODULE_NAME_DELIMETER), ipSubModules[i].Name); // Add the name of the module as a prefix to the name given in the declaration initialization
				END_IF
			END_IF
		END_FOR

		SequenceState := SequenceState + 10;

	20:
		NumberOfComponents := 0;
		FOR i := 1 TO Parameters_PackML_Base.MAX_NO_OF_COMPONENTS DO
			IF ipComponents[i] <> 0 THEN
				NumberOfComponents := NumberOfComponents + 1;
				IF Parameters_PackML_Base.CONCAT_COMPONENT_NAME_WITH_PARENT THEN
					ipComponents[i].Name := CONCAT(CONCAT(_Name, Parameters_PackML_Base.COMPONENT_NAME_DELIMETER), ipComponents[i].Name); // Add the name of the module as a prefix to the name given in the declaration initialization
				END_IF
			END_IF
		END_FOR

		SequenceState := SequenceState + 10;

	30:
		// Initialize subunit overview used by state machine
		PMLSubModuleInfoRef.ArraySize	 := SIZEOF(PMLSubModuleInfo);
		PMLSubModuleInfoRef.NoOfSubUnits := NumberOfSubModules;
		PMLSubModuleInfoRef.pArray		 := ADR(PMLSubModuleInfo);
		SequenceState					 := SequenceState + 10;

	40:
		// Initialization for this module is not complete until all subunits/components are finished
		// with their own Initialize().  This is called from CyclicLogic() so call from here until they are initialized.
		IF Parameters_PackML_Base.SUBSEQUENT_INIT_CALLS THEN
			IF m <= NumberOfSubModules THEN
				IF ipSubModules[m] <> 0 AND_THEN NOT ipSubModules[m].InitComplete THEN
					AllSubUnitsInitialized := FALSE;
					ipSubModules[m].CyclicLogic();
				ELSE
					m := m + 1;
				END_IF
			END_IF

			IF c <= NumberOfSubModules THEN
				IF ipComponents[c] <> 0 AND_THEN NOT ipComponents[c].InitComplete THEN
					AllComponentsInitialized := FALSE;
					ipComponents[c].CyclicLogic();
				ELSIF ipComponents[c] <> 0 AND_THEN ipComponents[c].InitComplete THEN
					c := c + 1;
				END_IF
			END_IF
		ELSE
			FOR i := 1 TO NumberOfSubModules DO
				IF ipSubModules[i] <> 0 AND_THEN NOT ipSubModules[i].InitComplete THEN
					AllSubUnitsInitialized := FALSE;
					ipSubModules[i].CyclicLogic();
				END_IF
			END_FOR

			FOR i := 1 TO NumberOfComponents DO
				IF ipComponents[i] <> 0 AND_THEN NOT ipComponents[i].InitComplete THEN
					AllComponentsInitialized := FALSE;
					ipComponents[i].CyclicLogic();
				END_IF
			END_FOR
		END_IF

		IF AllSubUnitsInitialized AND AllComponentsInitialized THEN
			SequenceState := 0;
			Initialize	  := TRUE;
		END_IF
END_CASE
END_METHOD

// Called one Cycle on State Change
METHOD PROTECTED ModeChanged
VAR_INPUT
END_VAR
END_METHOD

METHOD PROTECTED FINAL RegisterComponent
VAR_INPUT
	Component : I_ComponentBase;
END_VAR

VAR
	i		: UDINT;
	PLCStop : PLC_Stop;
END_VAR
IF NOT _InitComplete AND (Component <> 0) THEN
	FOR i := 1 TO Parameters_PackML_Base.MAX_NO_OF_COMPONENTS DO
		IF ipComponents[i] = Component THEN
			// Component already registered
			RETURN;
		END_IF
	END_FOR

	FOR i := 1 TO Parameters_PackML_Base.MAX_NO_OF_COMPONENTS DO
		IF ipComponents[i] = 0 THEN
			ipComponents[i] := Component;
			RETURN;
		END_IF
	END_FOR

	// If we get here then we are exceeding the array bounds
	Trace(CONCAT('***CRITICAL - Failed to register component!!  (', CONCAT(Component.Name, ')***')));
	PLCStop(STOP := TRUE);
END_IF
END_METHOD

METHOD FINAL RegisterExternalController : BOOL
VAR_INPUT
	Controller : I_PackML_ExternalController;
END_VAR

VAR
	i : UDINT;
END_VAR
FOR i := 1 TO Parameters_PackML_Base.MAX_NO_OF_EXTERNAL_CONTROLLERS DO
	IF ipExternalControllers[i] = 0 THEN
		ipExternalControllers[i]   := Controller;
		Controller.Control		   := THIS^;
		RegisterExternalController := TRUE;
		RETURN;
	END_IF
END_FOR

// If you get this far you have already registered the maximum number of controllers
RegisterExternalController := FALSE;
END_METHOD

METHOD PROTECTED FINAL RegisterSubmodule
VAR_INPUT
	SubModule : I_PackML_BaseModule;
END_VAR

VAR
	i		: UDINT;
	PLCStop : PLC_Stop;
END_VAR
IF NOT _InitComplete AND (SubModule <> 0) THEN
	FOR i := 1 TO Parameters_PackML_Base.MAX_NO_OF_SUBMODULES DO
		IF ipSubModules[i] = SubModule THEN
			// Submodule already registered
			RETURN;
		END_IF
	END_FOR

	FOR i := 1 TO Parameters_PackML_Base.MAX_NO_OF_SUBMODULES DO
		IF ipSubModules[i] = 0 THEN
			ipSubModules[i] := SubModule;
			RETURN;
		END_IF
	END_FOR

	// If we get here then we are exceeding the array bounds
	Trace(CONCAT('***CRITICAL - Failed to register SubModule!!  (', CONCAT(SubModule.Name, ')***')));
	PLCStop(STOP := TRUE);
END_IF
END_METHOD

// Called one Cycle on State Change
METHOD PROTECTED StateChanged
VAR_INPUT
END_VAR
END_METHOD

// Signals to the state manager FB when a state has completed
METHOD PROTECTED StateComplete

// This method is called by any of the transition state's logic methods as required
//*************************************************************************************************************************************************************************

// If you are about to write application specific code, note that any such code should exist within the "Application" directory using a Function Block that 'EXTENDS' this base Function Block!

// This particular method's functionality can be overriden in the extended block by creating a method of the same name, with desired functionality therein

// If the functionality of this base module is to be retained, but more functionality is desired, the extended method can contain a SUPER^.ThisMethodName(); call, which will call this code
//*************************************************************************************************************************************************************************
StateMachine.M_StateComplete();
END_METHOD

END_FUNCTION_BLOCK

// PackML/FB_PackML_StateLogger
// This FB raises events corresponding to state changes within the parent PackML module
FUNCTION_BLOCK FB_PackML_StateLogger
VAR_IN_OUT
	Alarms : ARRAY[1..48] OF FB_TcAlarm; // Array of alarms for Core PackML events that exist in any PackML enabled module
END_VAR

VAR_INPUT
	ModulePrefix  : STRING;		  // Prefix String for all state change events (Typically the ID and Name of the module in some concatenated form)
	State		  : E_PMLState;	  // Current PackML state of the module
	LogAllChanges : BOOL := TRUE; // If TRUE, all state change events will be logged, regardless of severity, otherwise info alarms are ignored
END_VAR

VAR
	LastState  : E_PMLState := E_PMLState.Aborted; // Saves the previous state each time the block is run
	pTempAlarm : REFERENCE TO FB_TcAlarm;		   // Temporary reference that makes severity checking simpler vs individually checking each change alarm within the case statement
END_VAR

IF State <> LastState THEN // If state has changed
	CASE State OF		   // Get the stored alarm that corresponds to the newly entered state and save its reference temporarily
		E_PMLState.Starting:
			pTempAlarm REF= Alarms[E_PackMLBase_Alarms.StateStartingEnter];

		E_PMLState.Execute:
			pTempAlarm REF= Alarms[E_PackMLBase_Alarms.StateExecuteEnter];

		E_PMLState.Completing:
			pTempAlarm REF= Alarms[E_PackMLBase_Alarms.StateCompletingEnter];

		E_PMLState.Completed:
			pTempAlarm REF= Alarms[E_PackMLBase_Alarms.StateCompleteEnter];

		E_PMLState.Resetting:
			pTempAlarm REF= Alarms[E_PackMLBase_Alarms.StateResettingEnter];

		E_PMLState.Idle:
			pTempAlarm REF= Alarms[E_PackMLBase_Alarms.StateIdleEnter];

		E_PMLState.Holding:
			pTempAlarm REF= Alarms[E_PackMLBase_Alarms.StateHoldingEnter];

		E_PMLState.Held:
			pTempAlarm REF= Alarms[E_PackMLBase_Alarms.StateHeldEnter];

		E_PMLState.Unholding:
			pTempAlarm REF= Alarms[E_PackMLBase_Alarms.StateUnholdingEnter];

		E_PMLState.Suspending:
			pTempAlarm REF= Alarms[E_PackMLBase_Alarms.StateSuspendingEnter];

		E_PMLState.Suspended:
			pTempAlarm REF= Alarms[E_PackMLBase_Alarms.StateSuspendedEnter];

		E_PMLState.Unsuspending:
			pTempAlarm REF= Alarms[E_PackMLBase_Alarms.StateUnsuspendingEnter];

		E_PMLState.Stopping:
			pTempAlarm REF= Alarms[E_PackMLBase_Alarms.StateStoppingEnter];

		E_PMLState.Stopped:
			pTempAlarm REF= Alarms[E_PackMLBase_Alarms.StateStoppedEnter];

		E_PMLState.Aborting:
			pTempAlarm REF= Alarms[E_PackMLBase_Alarms.StateAbortingEnter];

		E_PMLState.Aborted:
			pTempAlarm REF= Alarms[E_PackMLBase_Alarms.StateAbortedEnter];

		E_PMLState.Clearing:
			pTempAlarm REF= Alarms[E_PackMLBase_Alarms.StateClearingEnter];

		E_PMLState.Undefined:
			pTempAlarm REF= Alarms[E_PackMLBase_Alarms.StateUndefinedEnter];
	END_CASE

	// If the FB is set to log all changes, log the change, otherwise check the severity of the alarm and log it if it exceeds 'info' severity
	IF LogAllChanges OR (pTempAlarm.eSeverity <> TcEventSeverity.Info AND pTempAlarm.eSeverity <> TcEventSeverity.Verbose) THEN
		pTempAlarm.Raise(0);
	END_IF

	CASE LastState OF // Clear the previous state's event (Events will remain 'Raised' as long as the module remains in that state)
		E_PMLState.Starting:
			Alarms[E_PackMLBase_Alarms.StateStartingEnter].Clear(0, 0);

		E_PMLState.Execute:
			Alarms[E_PackMLBase_Alarms.StateExecuteEnter].Clear(0, 0);

